# B&R Automation Studio project TD52 (part 139)

#### Vent_ERCyclic.st
```iecst
(*******************************************************************************
Vent_ER			ventilation engine room

This code is confidential and proprietary to the INNIO Company.
It may not be used in any form, or reproduced in any manner,
without the express written permission of the INNIO Company.
Copyright, INNIO Company, 2019

Customized modifications: -
------------------------

History:
-------
V0.1	04.07.1998	Pa			erstellt
 		24.11.1998	Pa			korrekturlesung
V170	06.02.2002	LH			Erfassung Raumtemperatur
V172	02.07.2002	LH			Ventilatoransteuerung, Variante ohne Jalousien
V173	13.11.2002	LH			Einlesen des Analogeinganges in pb17 verlegt
V180	25.02.2003	LH			überarbeitet, Grenzwerte über Rezept
 								Notkühler --> Kühler und erweitert auf 4 Stufen
 								Gemischkühler neu und in 4 Stufen
V181	13.05.2003	LH			Initialisierung für Kühler (Schrittkette)
 		05.06.2003	LH			GW Raumtemperatur angepasst
 		24.06.2003	LH			Gemischkühler in 3 Stufen
V182	04.08.2003	LH			Erfassung Ansauglufttemperatur
V183	25.11.2003	LH			Gemischkühler wieder in 4 Stufen
 								Variante Kombikühler eingeführt
V184	12.01.2004	LH			Ventilation bei Messignal Raumtemperatur
V206	22.06.2004	LH			Raumlüftung NEU aufgrund von Synchronisierproblemen
V207	23.09.2004	LH			20 min. Nachlauf der geregelten Ventilation (Kruckenhauser)
 								Ansauglufttemperatur aktiviert
V2071	05.02.2005	LH			Aktivierung Messtelle Raumtemperatur über Parameter
 		23.02.2005	LH			Nachlauf der geregelten Ventilation nur mit Anforderung Hilfsbetriebe! (Egger)
V2073b	16.05.2006	LH			Lüftung 100% auch bei Gasalarm
V190	09.09.2004	LH			Raumtemperatur und Ansauglufttemperatur --> eigene tasks
 								Lüftung im Stillstand erst mit 40°C
V210	08.09.2004	LH			Variante Raumlüftung für kalte Länder
 								Initialisierung Kühlerschrittkette erweitert auf 11 Regler
 		16.11.2005	LH			Ansteuerung Frequenzumformer bei Gasvoralarm bzw. N2-Spuelung korrigiert
V230	24.01.2008	LH			wegen Einführung Gemischkühlerschrittkette 4-stufigen Gemischkühler gelöscht
V2.34.0	15.10.2008	lettenb.	M_NKWD replaced with M_NKWD_W
V3.10.0	17.02.2010	lettenb.	MRL_FU: EINS -> bAirInVentF(parameter) fehlerbehebung(bruno plattn.)
.								(W2120 störg.raumlüftg.kommt wenn keine raumlüftung)
V3.20.0	30.09.2010	maier(BuR)	M_GSEIN replaced with GCB_ON
.		17.12.2010	lettenb.	purge cycle added, K_var/K_anz/Anz_anfhbt/K_reg setting from parameter
V3.30.0	14.09.2011	lettenb.	FG_FU: dmnd_purge added (bugfix)
V3.99.0 15.02.2013	lettenb.	pb3_VE renamed to Vent_ER
V4.00.0	08.04.2015				FG_FU:(var.with louvers) Para.bER_VentColdCountryMode 'NOT' added(bugfix)
V4.02.0 03.08.2015  Stary       FG_FU: added variant with 2 controlled inlet+outlet louvers
		07.08.2015  Denk		Manual operating auxiliaries control functionality added
		13.08.2015	lettenb.	OUT_VE.tRel_ER_Fan.Do: var.for noFU added(undef.demand ZJAL2 with gcb.on/off)(hackel)
        09.12.2015  Stary       line 189-192: modified variable for louver feedback check
V4.04.0 20.05.2016	lettenb.	tDemPurgeER.Do added, bugfix
V4.04.0 27.09.2016  Stary       Task modified with introduction of cases for the variant-management engine room ventilation
		24.10.2016  Stary       changed parameters for release engine-room ventilation depending on analog position-feedback louvers - bugfix
		21.12.2016  Stary       modification of code after software-test on simulator
		23.01.2017  Stary       modification of code after test with WINMODE (bugfix)
		27.02.2017  Stary       added AND NOT IN_VE.bMsg1031 in release FC (bugfix)
		03.03.2017  lettenb.    added AND NOT IN_VE.bMsg1054 in release FC (bugfix)
		08.05.2017	lettenb.	FG_FU, tRel_ER_FC logic corr., bugfix
V4.05.0 20.09.2017	Messner		Active Cooling Program added
V4.07.0 25.02.2019	lettenb.	bERV_NotRdy engine room ventilation not ready - block engine start added, PWR-FFI-2018-0637 gem. TA 1100-0110
		13.05.2019	lettenb.	ANF_LUE: room vent.active with RTM40(not just minimum fan speed) and extended cooldown time after engine stop
		17.09.2019	lettenb.	ZJAL2: man.aux.control if only 1 inair louver is active, bugfix
V4.10.0	22.12.2020	lettenb.	config VAR.21/22: analog louvers with fix speed fans(set ZJAL1,ZJAL2,AJAL for this config.)
		25.01.2021	lettenb.	engine room ventilation not ready - block engine start: OUT_VE.bERV_NotRdy moved to task MsgVE, bugfix
V4.11.0	23.11.2021	lettenb.	processed signales to AuxRelEngOp (release engine operation) depending on louvers configuration, bugfix
V4.13.0 25.09.2023	Bacci		added IN_VE.tAuxV_Supply_Ok.Di in release FC
		05.12.2023	Bacci		Added ventilation demand before starting the ingition selftest and exhaust scavenging. New DO for inlet louvers demand for customer
V4.14.0 25.11.2024	Bacci		T6 Start procedure with purge start (2024-219): added ventilation demand before purge cranking cycle during fast start preparation
V4.25.0 26.11.2025	Bacci		Safety Function - Insufficient Ventilation (2024-202): reactivation of cold county function and safety plausibility check added

Instructions for use:
--------------------

Outstandings:
------------
*******************************************************************************)
PROGRAM _CYCLIC

	(* parameter *)
	Para.bLouvers;					(* engine room ventilation with louvers *)
	Para.bER_VentColdCountryMode;	(* engine room ventilation cold country mode *)
	Para.bVISA;						(* monitoring according VISA *)

	(*----------------------------------------------------------------------------------------------*)
	(* start ventilation *)
	RTM25 := bT_AirER_Hi1 OR IN_VE.tT_AirER_Ext_Hi1.Di OR IN_VE.bACP_AirER_Dem;

	(* ventilation stage 2 *)
	RTM30 := bT_AirER_Hi2 OR IN_VE.tT_AirER_Ext_Hi2.Di;

	(* start ventilation at stopped engine *)
	RTM40 := bT_AirER_Hi4 OR IN_VE.bACP_AirER_Dem;

	(* demand engine room ventilation for purge cycle *)
	dmnd_purge	:=	Para.bPurgecycle_Active
				AND(IN_VE.bEng_Dem OR IN_VE.bGV_On);

	OUT_VE.tDemPurgeER.Do := dmnd_purge;

	(* signal failure for engine room ventilation *)
	IF Para.bER_VentColdCountryMode THEN
		MS_LUE	:= (IN_VE.bAMM_T_Ch_T1LP_Avg AND IN_VE.bEng_Aux_Dem_CDR)
				OR  MM2VIS.bMsg3152;
	ELSE
		MS_LUE	:=  MM2VIS.bMsg3152;
	END_IF;

	(* purge cycle time *)
	xTON_purgecycle(IN:= OUT_VE.tRel_ER_FC.Do AND NOT MM2VIS.bMsg2120 AND NOT MM2VIS.bMsg2795 AND NOT MM2VIS.bMsg2796, PT:= T#60s);
	OUT_VE.bPurgeER_Rdy := IN_VE.tAirER_FS.Di AND xTON_purgecycle.Q;

	(* Demand engine room ventilation *)
	ANF_LUE	:= IN_VE.bEng_Aux_Dem_CDR
			OR dmnd_purge
			OR IN_VE.bACP_AirER_Dem
			OR RTM40;

	(* fan speed minimum *)
	OUT_VE.tSet_ER_Fan_Min.Do := (IN_VE.bEng_Aux_Dem OR dmnd_purge)
						  AND NOT IN_VE.tGCB_On.Di;

	(* release increased ventilation intensity *)
	IF Para.bInAirER_Fan_FU OR Para.bOutAirER_Fan_FU THEN
		OUT_VE.tRel_ER_Fan.Do := ANF_LUE AND NOT OUT_VE.tSet_ER_Fan_Min.Do;
	ELSE
		OUT_VE.tRel_ER_Fan.Do := ANF_LUE;
	END_IF;

	(* inlet louvers demand for customer. Ventilation in our scope *)
	OUT_VE.tDemERVentInLou_Cust.Do := IN_VE.bInLouDemIgn OR IN_VE.bInLouDemEX OR IN_VE.bInLouDemAG;

	IF IN_VE.bSafetyPLC_Active AND NOT Para.bSafe_ERV_Cust_Active THEN
		(* Cold country mode active for safety PLC *)
		OUT_VE.bERV_ColdCountry := Para.bER_VentColdCountryMode AND NOT (bT_InAirER_LimHi_Lou OR RTM40 OR MS_LUE);

		(*----------------------------------------------------------------*)
		(* safety plausibility check for inlet, outlet louvers and fans *)
		(*----------------------------------------------------------------*)
		(* Minimum release conditions for safety plausibility checks *)
		bRel_ERV_SafeCheck_Min := 	NOT IN_VE.bEng_Aux_Dem_CDR									(* CDR done*)
								AND NOT dmnd_purge												(* Engine room purge done *)
								AND NOT IN_VE.bInLouDemIgn										(* Ignition self test done*)
								AND NOT IN_VE.bInLouDemEX										(* Exhaust gas scavenging done *)
								AND NOT IN_VE.bInLouDemAG										(* Inlet louver demended for purge cycle during fast start preparation *)
								AND NOT (IN_VE.bInAirER_FanSet100 AND IN_VE.bRel_ScavN2)		(* Nitrogen scavenging done*)
								AND NOT IN_VE.bMsg1054											(* No fire alarm *)
								AND NOT IN_VE.bMsg1031											(* No emergency stop*)
								AND NOT IN_VE.bMsg1052											(* No gas prealarm *)
								AND NOT IN_VE.bMsg1053;											(* No gas alarm *)

		(* Extended release conditions for safety plausibility checks *)
		bRel_ERV_SafeCheck_Ext := 		bRel_ERV_SafeCheck_Min
								AND NOT MS_LUE										(* No engine room or engine intake temparture MSF *)
								AND NOT OUT_VE.bMsg2705								(* No engine room differential pressure MSF *)
								AND NOT RTM40										(* High engine room temperature at engine stop *)
								AND NOT IN_VE.tManAuxCtr.bInAirER_Lou1DemOpen 		(* No inlet louvers 1 manual request *)
								AND NOT IN_VE.tManAuxCtr.bInAirER_Lou2DemOpen		(* No inlet louvers 2 manual request *)
								AND NOT IN_VE.tManAuxCtr.bOutAirER_LouDemOpen		(* No outlet louvers manual request *)
								AND NOT IN_VE.tManAuxCtr.bER_FC_Set;				(* No ventilation fan frequency converter manual request *)

		(* engine stopped within 50 min *)
		xTOF_EngStop_SafeCheck(IN:= IN_VE.bEng_Aux_Dem_CDR, PT:= T#50m);

		(* reset plausibility check status *)
		xR_TRIG_bERV_SafeCheck_OK_Rset(CLK := IN_VE.bEng_Aux_Dem_CDR);
		IF xR_TRIG_bERV_SafeCheck_OK_Rset.Q THEN
			bERV_SafeCheck_OK := FALSE;
		END_IF;

		(* General release for safety plauibility checks *)
		bRel_ERV_SafeCheck := (bRel_ERV_SafeCheck_Ext OR (bRel_ERV_SafeCheck_Min AND (NOT xTOF_EngStop_SafeCheck.Q OR IN_VE.bERV_PC_Forced))) AND xOpMode.Stop;
		xR_TRIG_bRel_ERV_SafeCheck(CLK := bRel_ERV_SafeCheck);

		(* break safe plausibility check in case minimum release requirement not fulfilled or extended release not fulfilled while engine stopped within 50 minutes and no check force from safety PLC *)
		IF NOT bRel_ERV_SafeCheck THEN
			iStepCnt_SafeCheck := 0;
		(* activate safe plausibility check in case of extended release conditions fulfilled or minimum release condition fulfilled and engine stopped longer than 50 min or heck force from safety PLC *)
		ELSIF xR_TRIG_bRel_ERV_SafeCheck.Q AND NOT bERV_SafeCheck_OK THEN
			iStepCnt_SafeCheck := 10;
		END_IF;

		(*----------------------------------------------------------------*)
		IF iStepCnt_SafeCheck = 0 THEN
			bERV_SafeCheck_CloseLou	:= FALSE;
			bERV_SafeCheck_OpenLou	:= FALSE;
			OUT_VE.bERV_Lou_PC_OP	:= FALSE;
			OUT_VE.bERV_Lou_PC_CL 	:= FALSE;
			xTON_ERV_SafeCheck_CloseLou(IN:= FALSE, PT:= T#0s);
			xTON_ERV_SafeCheck_OpenLou(IN:= FALSE, PT:= T#0s);
		END_IF;

		(*----------------------------------------------------------------*)
		(* Step 1: close louvers for 3 minutes*)
		IF iStepCnt_SafeCheck = 10 THEN
			bERV_SafeCheck_CloseLou	:= TRUE;
			xTON_ERV_SafeCheck_CloseLou.IN := TRUE;
			xTON_ERV_SafeCheck_CloseLou.PT :=  T#180s;

			IF xTON_ERV_SafeCheck_CloseLou.Q THEN
				bERV_SafeCheck_CloseLou	:= FALSE;
				xTON_ERV_SafeCheck_CloseLou.IN := FALSE;
				xTON_ERV_SafeCheck_CloseLou.PT :=  T#0s;
				iStepCnt_SafeCheck := iStepCnt_SafeCheck + 10;
			END_IF;
		END_IF;
		(*----------------------------------------------------------------*)
		(* Step 2: open louvers for 3 minutes*)
		IF iStepCnt_SafeCheck = 20 THEN
			bERV_SafeCheck_OpenLou	:= TRUE;
			OUT_VE.bERV_Lou_PC_OP := TRUE;
			xTON_ERV_SafeCheck_OpenLou.IN := TRUE;
			xTON_ERV_SafeCheck_OpenLou.PT :=  T#180s;

			IF xTON_ERV_SafeCheck_OpenLou.Q THEN
				bERV_SafeCheck_OpenLou	:= FALSE;
				OUT_VE.bERV_Lou_PC_OP := FALSE;
				xTON_ERV_SafeCheck_OpenLou.IN := TRUE;
				xTON_ERV_SafeCheck_OpenLou.PT :=  T#0s;
				iStepCnt_SafeCheck := iStepCnt_SafeCheck + 10;
			END_IF;
		END_IF;

		(*----------------------------------------------------------------*)
		(* Step 3: close louvers for 3 minutes*)
		IF iStepCnt_SafeCheck = 30 THEN
			bERV_SafeCheck_CloseLou	:= TRUE;
			OUT_VE.bERV_Lou_PC_CL := TRUE;
			xTON_ERV_SafeCheck_CloseLou.IN := TRUE;
			xTON_ERV_SafeCheck_CloseLou.PT :=  T#180s;

			IF xTON_ERV_SafeCheck_CloseLou.Q THEN
				bERV_SafeCheck_CloseLou	:= FALSE;
				OUT_VE.bERV_Lou_PC_CL := FALSE;
				xTON_ERV_SafeCheck_CloseLou.IN := FALSE;
				xTON_ERV_SafeCheck_CloseLou.PT :=  T#0s;
				bERV_SafeCheck_OK := TRUE;
				iStepCnt_SafeCheck := 0;
			END_IF;
		END_IF;

		(*----------------------------------------------------------------*)
	ELSE
		OUT_VE.bERV_ColdCountry :=FALSE;
		bERV_SafeCheck_CloseLou := FALSE;
		bERV_SafeCheck_OpenLou := FALSE;
		OUT_VE.bERV_Lou_PC_OP := FALSE;
		OUT_VE.bERV_Lou_PC_CL := FALSE;
		xTON_ERV_SafeCheck_CloseLou(IN:= FALSE, PT:= T#0s);
		xTON_ERV_SafeCheck_OpenLou(IN:= FALSE, PT:= T#0s);
	END_IF;

		(* Call of the FUB *)
		xTON_ERV_SafeCheck_CloseLou();
		xTON_ERV_SafeCheck_OpenLou();

(*---------------------------------------------------------- INLET LOUVERS HANDLING -----------------------------------------------------------------------------------*)
// 	CONTROL-TYPE
	Para.iTypeCtr_InlLou_ERV; 		// (0-2)  0 ... no control of louvers
							  		//        1 ... engine room inlet louvers 1+2 demanded (DO)
							  		//        2 ... inlet louvers controlled (AO)
//	FEEDBACK-TYPE
	Para.iTypeFeedback_InlLou_ERV; 	// (0-2)  0 ... no feedback-signals
								   	//        1 ... feedback signals digital (DI)
								   	//        2 ... feedback signals analog (AI)

   	(* HANDLING OF CASES FOR RELEASE ROOM-VENTILATION *)
	iValueInlLou := Para.iTypeCtr_InlLou_ERV * 10 + Para.iTypeFeedback_InlLou_ERV; // according to this value the variants will run into the fitting case

	//		0 ... no control and no feedback
	//	   11 ... louvers demanded, feedback signal digital
	//     12 ... louvers demanded, feedback signal analog
	//     21 ... louvers controlled, feedback signal digital
	//     22 ... louvers controlled, feedback signal analog

	CASE iValueInlLou OF

	// ------------------------------------ no control and no feedback -----------------------------------------------------------------------
	  0:
		 	IN_VE.tInAirER_Lou1Opened.Di	:=	IN_VE.tInAirER_Lou1Opened.Di OR	NOT IN_VE.tInAirER_Lou1Opened.GoodQual;
			IN_VE.tInAirER_Lou2Opened.Di	:=	IN_VE.tInAirER_Lou2Opened.Di OR	NOT IN_VE.tInAirER_Lou2Opened.GoodQual;

			(* needed for demand air inlet fan 1 (fix-speed) *)
			ZJAL1 	:=(((bT_InAirER_LimHi_Lou OR NOT Para.bER_VentColdCountryMode) AND (IN_VE.bEng_Aux_Dem_CDR OR dmnd_purge))
					OR	RTM40
					OR	MS_LUE
					OR	IN_VE.bInLouDemIgn (* inlet louver demended for ignition self test *)
					OR	IN_VE.bInLouDemEX  (* inlet louver demended for scavenging *)
					OR	IN_VE.bInLouDemAG  (* inlet louver demended for purge cycle during fast start preparation *)
					OR (IN_VE.bInAirER_FanSet100 AND IN_VE.bRel_ScavN2)
					OR	bERV_SafeCheck_OpenLou) (* louver demand for safety plausibility check*)
					AND NOT bERV_SafeCheck_CloseLou; (* louver closed for safety plausibility check*)

			OUT_VE.tInAirER_Lou1DemOpen.Do	:= (ZJAL1 AND NOT IN_VE.bMsg1054 AND NOT IN_VE.bMsg1031)
											OR	IN_VE.bMsg1052
											OR	IN_VE.bMsg1053;

			(* needed for demand air inlet fan 2 (fix-speed) *)
			IF Para.bInAirER_Fan_FU THEN
				ZJAL2	:=(((bT_InAirER_LimHi_Lou OR NOT Para.bER_VentColdCountryMode) AND (IN_VE.bEng_Aux_Dem_CDR OR dmnd_purge))
						OR	RTM40
						OR	MS_LUE
						OR	IN_VE.bInLouDemIgn (* inlet louver demended for ignition self test *)
						OR	IN_VE.bInLouDemEX  (* inlet louver demended for scavenging *)
						OR	IN_VE.bInLouDemAG  (* inlet louver demended for purge cycle during fast start preparation *)
						OR (IN_VE.bInAirER_FanSet100 AND IN_VE.bRel_ScavN2)
						OR	bERV_SafeCheck_OpenLou) (* louver demand for safety plausibility check*)
						AND NOT bERV_SafeCheck_CloseLou; (* louver closed for safety plausibility check*)

			ELSE
				ZJAL2	:= ((RTM30 AND OUT_VE.tRel_ER_Fan.Do)
						OR	MS_LUE
						OR	IN_VE.bInLouDemIgn (* inlet louver demended for ignition self test *)
						OR	IN_VE.bInLouDemEX  (* inlet louver demended for scavenging *)
						OR	IN_VE.bInLouDemAG  (* inlet louver demended for purge cycle during fast start preparation *)
						OR (IN_VE.bInAirER_FanSet100 AND IN_VE.bRel_ScavN2)
						OR	bERV_SafeCheck_OpenLou) (* louver demand for safety plausibility check*)
						AND NOT bERV_SafeCheck_CloseLou; (* louver closed for safety plausibility check*)
			END_IF;

			OUT_VE.tInAirER_Lou2DemOpen.Do	:= (ZJAL2 AND NOT IN_VE.bMsg1054 AND NOT IN_VE.bMsg1031)
											OR	IN_VE.bMsg1052
											OR	IN_VE.bMsg1053;

			(* release engine room ventilation case 0 *)
			FG_FU_InlLou_Case0	:=	NOT IN_VE.bMsg1054
								AND NOT IN_VE.bMsg1031
								AND	  (((bOMSS_MAT AND IN_VE.bEng_Aux_Dem_CDR)
									OR (bOMSS_MAT AND dmnd_purge)
									OR (bOMSS_MAT AND RTM40)
									OR (bOMSS_MAT AND MM2VIS.bMsg3152)
									OR (IN_VE.bRel_ScavN2 AND IN_VE.bInAirER_FanSet100)
									OR  IN_VE.tManAuxCtr.bER_FC_Set)(* Manual operating auxiliaries control - Handbedienebene *)
									AND NOT bERV_SafeCheck_CloseLou) (* louver /fan off for safety plausibility check*)
									OR IN_VE.bMsg1052
									OR IN_VE.bMsg1053;

	// ------------------------------------- louvers demanded, feedback signal digital -------------------------------------------------------
	 11:
		    (* demand engine room air inlet louver 1 *)
	     	ZJAL1 	:=(((bT_InAirER_LimHi_Lou OR NOT Para.bER_VentColdCountryMode) AND (IN_VE.bEng_Aux_Dem_CDR OR dmnd_purge))
					OR	RTM40
					OR	MS_LUE
					OR (IN_VE.bInAirER_FanSet100 AND IN_VE.bRel_ScavN2)
					OR	IN_VE.bInLouDemIgn (* inlet louver demended for ignition self test *)
					OR	IN_VE.bInLouDemEX  (* inlet louver demended for scavenging *)
					OR	IN_VE.bInLouDemAG  (* inlet louver demended for purge cycle during fast start preparation *)
					OR  IN_VE.tManAuxCtr.bInAirER_Lou1DemOpen			(* Manual operating auxiliaries control - Handbedienebene *)
					OR	bERV_SafeCheck_OpenLou) (* louver demand for safety plausibility check*)
					AND NOT bERV_SafeCheck_CloseLou; (* louver closed for safety plausibility check*)

		 	OUT_VE.tInAirER_Lou1DemOpen.Do	:= (ZJAL1 AND NOT IN_VE.bMsg1054 AND NOT IN_VE.bMsg1031)
											OR	IN_VE.bMsg1052
											OR	IN_VE.bMsg1053;

			(* demand engine room air inlet louver 2 *)
			IF Para.bInAirER_Fan_FU THEN
				ZJAL2	:=(((bT_InAirER_LimHi_Lou OR NOT Para.bER_VentColdCountryMode) AND (IN_VE.bEng_Aux_Dem_CDR OR dmnd_purge))
						OR	RTM40
						OR	MS_LUE
						OR (IN_VE.bInAirER_FanSet100 AND IN_VE.bRel_ScavN2)
						OR	IN_VE.bInLouDemIgn (* inlet louver demended for ignition self test *)
						OR	IN_VE.bInLouDemEX  (* inlet louver demended for scavenging *)
						OR	IN_VE.bInLouDemAG  (* inlet louver demended for purge cycle during fast start preparation *)
						OR (IN_VE.tManAuxCtr.bInAirER_Lou1DemOpen AND NOT Para.bInAirER_Lou2_visible)	(* only 1 inlet louver active *)
						OR  IN_VE.tManAuxCtr.bInAirER_Lou2DemOpen			(* Manual operating auxiliaries control - Handbedienebene *)
						OR	bERV_SafeCheck_OpenLou) (* louver demand for safety plausibility check*)
						AND NOT bERV_SafeCheck_CloseLou; (* louver closed for safety plausibility check*)
			ELSE
				ZJAL2	:= ((RTM30 AND OUT_VE.tRel_ER_Fan.Do)
						OR	MS_LUE
						OR (IN_VE.bInAirER_FanSet100 AND IN_VE.bRel_ScavN2)
						OR	IN_VE.bInLouDemIgn (* inlet louver demended for ignition self test *)
						OR	IN_VE.bInLouDemEX  (* inlet louver demended for scavenging *)
						OR	IN_VE.bInLouDemAG  (* inlet louver demended for purge cycle during fast start preparation *)
						OR (IN_VE.tManAuxCtr.bInAirER_Lou1DemOpen AND NOT Para.bInAirER_Lou2_visible)	(* only 1 inlet louver active *)
						OR  IN_VE.tManAuxCtr.bInAirER_Lou2DemOpen			(* Manual operating auxiliaries control - Handbedienebene *)
						OR	bERV_SafeCheck_OpenLou) (* louver demand for safety plausibility check*)
						AND NOT bERV_SafeCheck_CloseLou; (* louver closed for safety plausibility check*)
			END_IF;

			OUT_VE.tInAirER_Lou2DemOpen.Do	:= (ZJAL2 AND NOT IN_VE.bMsg1054 AND NOT IN_VE.bMsg1031)
											OR	IN_VE.bMsg1052
											OR	IN_VE.bMsg1053;

			(* release engine room ventilation case 11 *)
			IN_VE.tInAirER_Lou2Opened.Di	:=	IN_VE.tInAirER_Lou2Opened.Di OR	NOT IN_VE.tInAirER_Lou2Opened.GoodQual;

			FG_FU_InlLou_Case11 := OUT_VE.tInAirER_Lou1DemOpen.Do AND IN_VE.tInAirER_Lou1Opened.Di
						       AND OUT_VE.tInAirER_Lou2DemOpen.Do AND IN_VE.tInAirER_Lou2Opened.Di;

			FG_InlVent_Step1_CtrInlLou := FALSE; // for correct case-change
			FG_InlVent_Step2_CtrInlLou := FALSE; // for correct case-change

	// ----------------------------------------- louvers demanded, feedback signal analog ----------------------------------------------------
	 12:
			(* demand engine room air inlet louver 1 *)
			ZJAL1 	:=(((bT_InAirER_LimHi_Lou OR NOT Para.bER_VentColdCountryMode) AND (IN_VE.bEng_Aux_Dem_CDR OR dmnd_purge))
					OR	RTM40
					OR	MS_LUE
					OR (IN_VE.bInAirER_FanSet100 AND IN_VE.bRel_ScavN2)
					OR	IN_VE.bInLouDemIgn (* inlet louver demended for ignition self test *)
					OR	IN_VE.bInLouDemEX  (* inlet louver demended for scavenging *)
					OR	IN_VE.bInLouDemAG  (* inlet louver demended for purge cycle during fast start preparation *)
					OR  IN_VE.tManAuxCtr.bInAirER_Lou1DemOpen			(* Manual operating auxiliaries control - Handbedienebene *)
					OR	bERV_SafeCheck_OpenLou) (* louver demand for safety plausibility check*)
					AND NOT bERV_SafeCheck_CloseLou; (* louver closed for safety plausibility check*)

			OUT_VE.tInAirER_Lou1DemOpen.Do	:= (ZJAL1 AND NOT IN_VE.bMsg1054 AND NOT IN_VE.bMsg1031)
											OR	IN_VE.bMsg1052
											OR	IN_VE.bMsg1053;

			(* demand engine room air inlet louver 2 *)
			IF Para.bInAirER_Fan_FU THEN
				ZJAL2	:=(((bT_InAirER_LimHi_Lou OR NOT Para.bER_VentColdCountryMode) AND (IN_VE.bEng_Aux_Dem_CDR OR dmnd_purge))
						OR	RTM40
						OR	MS_LUE
						OR (IN_VE.bInAirER_FanSet100 AND IN_VE.bRel_ScavN2)
						OR	IN_VE.bInLouDemIgn (* inlet louver demended for ignition self test *)
						OR	IN_VE.bInLouDemEX  (* inlet louver demended for scavenging *)
						OR	IN_VE.bInLouDemAG  (* inlet louver demended for purge cycle during fast start preparation *)
						OR (IN_VE.tManAuxCtr.bInAirER_Lou1DemOpen AND NOT Para.bInAirER_Lou2_visible)	(* only 1 inlet louver active *)
						OR  IN_VE.tManAuxCtr.bInAirER_Lou2DemOpen			(* Manual operating auxiliaries control - Handbedienebene *)
						OR	bERV_SafeCheck_OpenLou) (* louver demand for safety plausibility check*)
						AND NOT bERV_SafeCheck_CloseLou; (* louver closed for safety plausibility check*)
			ELSE
				ZJAL2	:= ((RTM30 AND OUT_VE.tRel_ER_Fan.Do)
						OR	MS_LUE
						OR (IN_VE.bInAirER_FanSet100 AND IN_VE.bRel_ScavN2)
						OR	IN_VE.bInLouDemIgn (* inlet louver demended for ignition self test *)
						OR	IN_VE.bInLouDemEX  (* inlet louver demended for scavenging *)
						OR	IN_VE.bInLouDemAG  (* inlet louver demended for purge cycle during fast start preparation *)
						OR (IN_VE.tManAuxCtr.bInAirER_Lou1DemOpen AND NOT Para.bInAirER_Lou2_visible)	(* only 1 inlet louver active *)
						OR  IN_VE.tManAuxCtr.bInAirER_Lou2DemOpen			(* Manual operating auxiliaries control - Handbedienebene *)
						OR	bERV_SafeCheck_OpenLou) (* louver demand for safety plausibility check*)
						AND NOT bERV_SafeCheck_CloseLou; (* louver closed for safety plausibility check*)
			END_IF;

			OUT_VE.tInAirER_Lou2DemOpen.Do	:= (ZJAL2 AND NOT IN_VE.bMsg1054 AND NOT IN_VE.bMsg1031)
											OR	IN_VE.bMsg1052
											OR	IN_VE.bMsg1053;

			(* check of position from inlet-louvers *)
			xGR_MAXR_InlLou1(In := IN_VE.tPos_InlLou1.Ai, Gw := Para.rPosLim_InlLou_Rel_ERV, Hy := Para.rPosLim_InlLou_Rel_ERV_Hy);
			xGR_MAXR_InlLou2(In := IN_VE.tPos_InlLou2.Ai, Gw := Para.rPosLim_InlLou_Rel_ERV, Hy := Para.rPosLim_InlLou_Rel_ERV_Hy);

			Pos_InlLou1_OK := Para.bPos_InlLou1_Active AND xGR_MAXR_InlLou1.Q;
			Pos_InlLou2_OK := Para.bPos_InlLou2_Active AND xGR_MAXR_InlLou2.Q;
			OUT_VE.Pos_InlLou1_OK := Pos_InlLou1_OK; // for release auxiliaries --> monitoring A1129 (AG)
			OUT_VE.Pos_InlLou2_OK := Pos_InlLou2_OK; // for release auxiliaries --> monitoring A1129 (AG)

			(* release engine room ventilation case 12 *)
			FG_FU_InlLou_Case12   := (OUT_VE.tInAirER_Lou1DemOpen.Do AND Pos_InlLou1_OK)
								AND ((OUT_VE.tInAirER_Lou2DemOpen.Do AND Pos_InlLou2_OK) OR NOT Para.bPos_InlLou2_Active);

			FG_InlVent_Step1_CtrInlLou := FALSE; // for correct case-change
			FG_InlVent_Step2_CtrInlLou := FALSE; // for correct case-change

	// -------------------------------------- louvers controlled, feedback signal digital --------------------------------------------------------------------
	 21:
			(* demand engine room air inlet louver *)
			ZJAL1 	:=((IN_VE.bEng_Aux_Dem_CDR OR dmnd_purge)
					OR	RTM40
					OR	MS_LUE
					OR (IN_VE.bInAirER_FanSet100 AND IN_VE.bRel_ScavN2)
					OR	bERV_SafeCheck_OpenLou) (* louver demand for safety plausibility check*)
					AND NOT bERV_SafeCheck_CloseLou; (* louver closed for safety plausibility check*)
					(*OUT_IG.bInLouDemIgn AND OUT_IG.bInLouDemEX AND IN_VE.bInLouDemAG not needed for fan activation. Louver AO signal defined in the Ctr_InlLou*)

			ZJAL2	:= ((RTM30 AND OUT_VE.tRel_ER_Fan.Do)
					OR	MS_LUE
					OR (IN_VE.bInAirER_FanSet100 AND IN_VE.bRel_ScavN2)
					OR	bERV_SafeCheck_OpenLou) (* louver demand for safety plausibility check*)
					AND NOT bERV_SafeCheck_CloseLou; (* louver closed for safety plausibility check*)

			(* release engine room ventilation case 21 *)
			IN_VE.tInAirER_Lou2Opened.Di := IN_VE.tInAirER_Lou2Opened.Di OR	NOT IN_VE.tInAirER_Lou2Opened.GoodQual;

			FG_FU_InlLou_Case21   := Para.bCtr_InlLou AND IN_VE.tInAirER_Lou1Opened.Di AND IN_VE.tInAirER_Lou2Opened.Di;

			(* air inlet fan 1 *)
			Release_InlVent_Step1_INT := (ZJAL1 AND NOT IN_VE.bMsg1054 AND NOT IN_VE.bMsg1031)  // general release ventilation step 1 depending on temperature, gas-alarm etc.
									OR	IN_VE.bMsg1052
									OR	IN_VE.bMsg1053;
			FG_InlVent_Step1_CtrInlLou := Release_InlVent_Step1_INT AND Para.bCtr_InlLou AND IN_VE.tInAirER_Lou1Opened.Di; 	// fix-speed inlet-fan 1

			(* air inlet fan 2 *)
			Release_InlVent_Step2_INT := (ZJAL2 AND NOT IN_VE.bMsg1054 AND NOT IN_VE.bMsg1031)  // general release ventilation step 2 depending on temperature, gas-alarm etc.
									OR	IN_VE.bMsg1052
									OR	IN_VE.bMsg1053;
			FG_InlVent_Step2_CtrInlLou := Release_InlVent_Step2_INT AND Para.bCtr_InlLou AND IN_VE.tInAirER_Lou1Opened.Di AND IN_VE.tInAirER_Lou2Opened.Di;  // fix-speed inlet-fan 2

			OUT_VE.tInAirER_Lou1DemOpen.Do := FALSE; // for correct case-change
			OUT_VE.tInAirER_Lou2DemOpen.Do := FALSE; // for correct case-change

	// --------------------------------------- louvers controlled, feedback signal analog ---------------------------------------------------------------------
	 22:
			(* demand engine room air inlet louver *)
			ZJAL1 	:=((IN_VE.bEng_Aux_Dem_CDR OR dmnd_purge)
					OR	RTM40
					OR	MS_LUE
					OR (IN_VE.bInAirER_FanSet100 AND IN_VE.bRel_ScavN2)
					OR	bERV_SafeCheck_OpenLou) (* louver demand for safety plausibility check*)
					AND NOT bERV_SafeCheck_CloseLou; (* louver closed for safety plausibility check*)
					(*OUT_IG.bInLouDemIgn AND OUT_IG.bInLouDemEX AND IN_VE.bInLouDemAG not needed for fan activation. Louver AO signalo defined in the Ctr_InlLou*)

			ZJAL2	:= ((RTM30 AND OUT_VE.tRel_ER_Fan.Do)
					OR	MS_LUE
					OR (IN_VE.bInAirER_FanSet100 AND IN_VE.bRel_ScavN2)
					OR	bERV_SafeCheck_OpenLou) (* louver demand for safety plausibility check*)
					AND NOT bERV_SafeCheck_CloseLou; (* louver closed for safety plausibility check*)

			(* check of position from inlet-louvers *)
			xGR_MAXR_InlLou1(In := IN_VE.tPos_InlLou1.Ai, Gw := Para.rPosLim_InlLou_Rel_ERV, Hy := Para.rPosLim_InlLou_Rel_ERV_Hy);
			xGR_MAXR_InlLou2(In := IN_VE.tPos_InlLou2.Ai, Gw := Para.rPosLim_InlLou_Rel_ERV, Hy := Para.rPosLim_InlLou_Rel_ERV_Hy);

			Pos_InlLou1_OK := Para.bPos_InlLou1_Active AND xGR_MAXR_InlLou1.Q;
			Pos_InlLou2_OK := Para.bPos_InlLou2_Active AND xGR_MAXR_InlLou2.Q;
			OUT_VE.Pos_InlLou1_OK := Pos_InlLou1_OK; // for release auxiliaries --> monitoring A1129 (AG)
			OUT_VE.Pos_InlLou2_OK := Pos_InlLou2_OK; // for release auxiliaries --> monitoring A1129 (AG)

			(* release engine room ventilation CASE 22 *)
			FG_FU_InlLou_Case22   := Para.bCtr_InlLou AND Pos_InlLou1_OK AND (Pos_InlLou2_OK OR NOT Para.bPos_InlLou2_Active);

			(* air inlet fan 1 *)
			Release_InlVent_Step1_INT := (ZJAL1 AND NOT IN_VE.bMsg1054 AND NOT IN_VE.bMsg1031)  // general release ventilation step 1 depending on temperature, gas-alarm etc.
									OR	IN_VE.bMsg1052
									OR	IN_VE.bMsg1053;
			FG_InlVent_Step1_CtrInlLou := Release_InlVent_Step1_INT AND Para.bCtr_InlLou AND Pos_InlLou1_OK;  // fix-speed inlet-fan 1

			(* air inlet fan 2 *)
			Release_InlVent_Step2_INT := (ZJAL2 AND NOT IN_VE.bMsg1054 AND NOT IN_VE.bMsg1031)  // general release ventilation step 2 depending on temperature, gas-alarm etc.
									OR	IN_VE.bMsg1052
									OR	IN_VE.bMsg1053;
			FG_InlVent_Step2_CtrInlLou := Release_InlVent_Step2_INT AND Para.bCtr_InlLou AND Pos_InlLou1_OK AND (Pos_InlLou2_OK OR NOT Para.bPos_InlLou2_Active);  // fix-speed inlet-fan 2

			OUT_VE.tInAirER_Lou1DemOpen.Do := FALSE; // for correct case-change
			OUT_VE.tInAirER_Lou2DemOpen.Do := FALSE; // for correct case-change

	END_CASE;

(*---------------------------------------------------------- OUTLET LOUVERS HANDLING -----------------------------------------------------------------------------------*)
// 	CONTROL-TYPE
	Para.iTypeCtr_OutlLou_ERV; 		// (0-2)  0 ... no control of louvers
							   		//        1 ... engine room outlet louvers 1+2 demanded (DO)
							   		//        2 ... outlet louvers controlled (AO)
//	FEEDBACK-TYPE
	Para.iTypeFeedback_OutlLou_ERV; // (0-2)  0 ... no feedback-signals
									//        1 ... feedback signals digital (DI)
									//        2 ... feedback signals analog (AI)

	(* HANDLING OF CASES FOR RELEASE ROOM-VENTILATION *)
	iValueOutlLou := Para.iTypeCtr_OutlLou_ERV*10 + Para.iTypeFeedback_OutlLou_ERV; // according to this value the variants will run into the fitting case

	//		0 ... no control and no feedback
	//	   11 ... louvers demanded, feedback signal digital
	//     12 ... louvers demanded, feedback signal analog
	//     21 ... louvers controlled, feedback signal digital
	//     22 ... louvers controlled, feedback signal analog

	CASE iValueOutlLou OF

		// --------------------------------------- no control and no feedback ------------------------------------------------------------
		0:
				IN_VE.tOutAirER_LouOpened.Di := IN_VE.tOutAirER_LouOpened.Di OR	NOT IN_VE.tOutAirER_LouOpened.GoodQual;

				(* needed for demand air inlet fan 1+2 (fix-speed) *)
				AJAL	:=	(IN_VE.bEng_Aux_Dem_CDR
						OR	dmnd_purge
						OR	RTM40
						OR	MS_LUE
						OR (IN_VE.bInAirER_FanSet100 AND IN_VE.bRel_ScavN2)
						OR	bERV_SafeCheck_OpenLou) (* louver demand for safety plausibility check*)
						AND NOT bERV_SafeCheck_CloseLou; (* louver closed for safety plausibility check*)

				OUT_VE.tOutAirER_LouDemOpen.Do	:= (AJAL AND NOT IN_VE.bMsg1031 AND NOT IN_VE.bMsg1054)
												OR	IN_VE.bMsg1052
												OR	IN_VE.bMsg1053;

				(* release engine room ventilation case 0 *)
				FG_FU_OutLou_Case0	:=	NOT IN_VE.bMsg1054
									AND NOT IN_VE.bMsg1031
									AND	  (((bOMSS_MAT AND IN_VE.bEng_Aux_Dem_CDR)
										OR (bOMSS_MAT AND dmnd_purge)
										OR (bOMSS_MAT AND RTM40)
										OR (bOMSS_MAT AND MM2VIS.bMsg3152)
										OR (IN_VE.bRel_ScavN2 AND IN_VE.bInAirER_FanSet100)
										OR  IN_VE.tManAuxCtr.bER_FC_Set) (* Manual operating auxiliaries control - Handbedienebene *)
										AND NOT bERV_SafeCheck_CloseLou) (* louver /fan off for safety plausibility check*)
										OR IN_VE.bMsg1052
										OR IN_VE.bMsg1053;

	// ---------------------------------------louvers demanded, feedback signal digital -----------------------------------------------------------
		11:
				(* demand engine room air outlet louvers *)
				AJAL	:=	(IN_VE.bEng_Aux_Dem_CDR
						OR	dmnd_purge
						OR	RTM40
						OR	MS_LUE
						OR (IN_VE.bInAirER_FanSet100 AND IN_VE.bRel_ScavN2)
						OR  IN_VE.tManAuxCtr.bOutAirER_LouDemOpen			(* Manual operating auxiliaries control - Handbedienebene *)
						OR	bERV_SafeCheck_OpenLou) (* louver demand for safety plausibility check*)
						AND NOT bERV_SafeCheck_CloseLou; (* louver closed for safety plausibility check*)

				OUT_VE.tOutAirER_LouDemOpen.Do	:= (AJAL AND NOT IN_VE.bMsg1031 AND NOT IN_VE.bMsg1054)
												OR	IN_VE.bMsg1052
												OR	IN_VE.bMsg1053;

				(* Release engine room ventilation case 12 *)
				FG_FU_OutlLou_Case11 := OUT_VE.tOutAirER_LouDemOpen.Do AND IN_VE.tOutAirER_LouOpened.Di;

				FG_InlVent_Step12_CtrOutlLou := FALSE; // for correct case-change

	// ---------------------------------------- louvers demanded, feedback signal analog -----------------------------------------------------------
		12:
				(* demand engine room air outlet louvers *)
				AJAL	:=	(IN_VE.bEng_Aux_Dem_CDR
						OR	dmnd_purge
						OR	RTM40
						OR	MS_LUE
						OR (IN_VE.bInAirER_FanSet100 AND IN_VE.bRel_ScavN2)
						OR  IN_VE.tManAuxCtr.bOutAirER_LouDemOpen			(* Manual operating auxiliaries control - Handbedienebene *)
						OR	bERV_SafeCheck_OpenLou) (* louver demand for safety plausibility check*)
						AND NOT bERV_SafeCheck_CloseLou; (* louver closed for safety plausibility check*)

				OUT_VE.tOutAirER_LouDemOpen.Do	:= (AJAL AND NOT IN_VE.bMsg1031 AND NOT IN_VE.bMsg1054)
												OR	IN_VE.bMsg1052
												OR	IN_VE.bMsg1053;

				(* check of position from outlet-louvers *)
				xGR_MAXR_OutlLou1(In:= IN_VE.tPos_OutlLou1.Ai, Gw:= Para.rPosLim_OutlLou_Rel_ERV, Hy:= Para.rPosLim_OutlLou_Rel_ERV_Hy);
				xGR_MAXR_OutlLou2(In:= IN_VE.tPos_OutlLou2.Ai, Gw:= Para.rPosLim_OutlLou_Rel_ERV, Hy:= Para.rPosLim_OutlLou_Rel_ERV_Hy);

				Pos_OutlLou1_OK := Para.bPos_OutlLou1_Active AND xGR_MAXR_OutlLou1.Q;
				Pos_OutlLou2_OK := Para.bPos_OutlLou2_Active AND xGR_MAXR_OutlLou2.Q;
				OUT_VE.Pos_OutlLou1_OK := Pos_OutlLou1_OK; // for release auxiliaries --> monitoring A1129 (AG)
				OUT_VE.Pos_OutlLou2_OK := Pos_OutlLou2_OK; // for release auxiliaries --> monitoring A1129 (AG)

				(* release engine room ventilation case 12 *)
				FG_FU_OutlLou_Case12	:= OUT_VE.tOutAirER_LouDemOpen.Do AND Pos_OutlLou1_OK AND (Pos_OutlLou2_OK OR NOT Para.bPos_OutlLou2_Active);

				FG_InlVent_Step12_CtrOutlLou := FALSE; // for correct case-change

	// ------------------------------------------- louvers controlled, feedback signal digital ---------------------------------------------------------
		21:
				(* demand air inlet fan 1+2 (fix-speed) *)
				AJAL	:=	(IN_VE.bEng_Aux_Dem_CDR
						OR	dmnd_purge
						OR	RTM40
						OR	MS_LUE
						OR (IN_VE.bInAirER_FanSet100 AND IN_VE.bRel_ScavN2)
						OR	bERV_SafeCheck_OpenLou) (* louver demand for safety plausibility check*)
						AND NOT bERV_SafeCheck_CloseLou; (* louver closed for safety plausibility check*)

				(* release engine room ventilation case 21 *)
				FG_FU_OutlLou_Case21	:= (Para.bCtr_OutlLou_RDP OR Para.bCtr_OutlLou_RT) AND IN_VE.tOutAirER_LouOpened.Di;

				(* air inlet fan 1+2 *)
			    Release_InlVent_StepINT	:= (AJAL AND NOT IN_VE.bMsg1031 AND NOT IN_VE.bMsg1054)	// general release ventilation step 1 depending on temperature, gas-alarm etc.
										OR	IN_VE.bMsg1052
										OR	IN_VE.bMsg1053;
				FG_InlVent_Step12_CtrOutlLou := Release_InlVent_StepINT AND (Para.bCtr_OutlLou_RDP OR Para.bCtr_OutlLou_RT) AND IN_VE.tOutAirER_LouOpened.Di;  // fix-speed inlet-fan 1+2

				OUT_VE.tOutAirER_LouDemOpen.Do := FALSE; // for correct case-change

	// -------------------------------------------- louvers controlled, feedback signal analog ---------------------------------------------------------
		22:
				(* demand air inlet fan 1+2 (fix-speed) *)
				AJAL	:=	(IN_VE.bEng_Aux_Dem_CDR
						OR	dmnd_purge
						OR	RTM40
						OR	MS_LUE
						OR (IN_VE.bInAirER_FanSet100 AND IN_VE.bRel_ScavN2)
						OR	bERV_SafeCheck_OpenLou) (* louver demand for safety plausibility check*)
						AND NOT bERV_SafeCheck_CloseLou; (* louver closed for safety plausibility check*)

				(* check of position from outlet-louvers *)
				xGR_MAXR_OutlLou1(In:= IN_VE.tPos_OutlLou1.Ai, Gw:= Para.rPosLim_OutlLou_Rel_ERV, Hy:= Para.rPosLim_OutlLou_Rel_ERV_Hy);
				xGR_MAXR_OutlLou2(In:= IN_VE.tPos_OutlLou2.Ai, Gw:= Para.rPosLim_OutlLou_Rel_ERV, Hy:= Para.rPosLim_OutlLou_Rel_ERV_Hy);

				Pos_OutlLou1_OK := Para.bPos_OutlLou1_Active AND xGR_MAXR_OutlLou1.Q;
				Pos_OutlLou2_OK := Para.bPos_OutlLou2_Active AND xGR_MAXR_OutlLou2.Q;
				OUT_VE.Pos_OutlLou1_OK := Pos_OutlLou1_OK; // for release auxiliaries --> monitoring A1129 (AG)
				OUT_VE.Pos_OutlLou2_OK := Pos_OutlLou2_OK; // for release auxiliaries --> monitoring A1129 (AG)

				(* release engine room ventilation CASE 22 *)
				FG_FU_OutlLou_Case22	:= (Para.bCtr_OutlLou_RDP OR Para.bCtr_OutlLou_RT) AND Pos_OutlLou1_OK AND (Pos_OutlLou2_OK OR NOT Para.bPos_OutlLou2_Active);

				(* air inlet fan 1+2 *)
				Release_InlVent_StepINT	:= (AJAL AND NOT IN_VE.bMsg1031 AND NOT IN_VE.bMsg1054)	// general release ventilation step 1 depending on temperature, gas-alarm etc.
										OR	IN_VE.bMsg1052
										OR	IN_VE.bMsg1053;
				FG_InlVent_Step12_CtrOutlLou := Release_InlVent_StepINT AND (Para.bCtr_OutlLou_RDP OR Para.bCtr_OutlLou_RT)
											AND Pos_OutlLou1_OK AND (Pos_OutlLou2_OK OR NOT Para.bPos_OutlLou2_Active);	// fix-speed inlet-fan 1+2

				OUT_VE.tOutAirER_LouDemOpen.Do := FALSE; // for correct case-change

	END_CASE;

(*------------------------ CASE CHECK FOR RELEASE ENGINE ROOM VENTILATION -----------------------------------------*)
	(* Inlet ventilation *)
	FG_FU_InlLou_ZW := (FG_FU_InlLou_Case0  AND iValueInlLou = 0)
					OR (FG_FU_InlLou_Case11 AND iValueInlLou = 11)
					OR (FG_FU_InlLou_Case12 AND iValueInlLou = 12)
					OR (FG_FU_InlLou_Case21 AND iValueInlLou = 21)
					OR (FG_FU_InlLou_Case22 AND iValueInlLou = 22);

	(* Outlet ventilation *)
	FG_FU_OutlLou_ZW := (FG_FU_OutLou_Case0  AND iValueOutlLou = 0)
					 OR (FG_FU_OutlLou_Case11 AND iValueOutlLou = 11)
					 OR (FG_FU_OutlLou_Case12 AND iValueOutlLou = 12)
					 OR (FG_FU_OutlLou_Case21 AND iValueOutlLou = 21)
					 OR (FG_FU_OutlLou_Case22 AND iValueOutlLou = 22);

(*---------------------------------------------------------- ROOM VENTILATION FAN HANDLING -----------------------------------------------------------------------------------*)

		(* air inlet fan 1 *)
		OUT_VE.tInAirER_Fan1DemOn.Do :=	(((OUT_VE.tInAirER_Lou1DemOpen.Do OR IN_VE.tManAuxCtr.bInAirER_Fan1DemOn) AND IN_VE.tInAirER_Lou1Opened.Di) OR FG_InlVent_Step1_CtrInlLou)
									AND (((OUT_VE.tOutAirER_LouDemOpen.Do OR IN_VE.tManAuxCtr.bInAirER_Fan1DemOn) AND IN_VE.tOutAirER_LouOpened.Di) OR FG_InlVent_Step12_CtrOutlLou);

		(* air inlet fan 2 *)
		OUT_VE.tInAirER_Fan2DemOn.Do := (((OUT_VE.tInAirER_Lou2DemOpen.Do OR IN_VE.tManAuxCtr.bInAirER_Fan2DemOn) AND IN_VE.tInAirER_Lou2Opened.Di) OR FG_InlVent_Step2_CtrInlLou)
									AND (((OUT_VE.tOutAirER_LouDemOpen.Do OR IN_VE.tManAuxCtr.bInAirER_Fan2DemOn) AND IN_VE.tOutAirER_LouOpened.Di) OR FG_InlVent_Step12_CtrOutlLou);

		(* release frequency converter for engine room ventilation (inlet/outlet) *)

		IF IN_VE.tManAuxCtr.bER_FC_Set THEN				(* Manual operating auxiliaries control - Handbedienebene *)
			FG_FU	:=	NOT IN_VE.bMsg1031
					AND NOT IN_VE.bMsg1054
					AND		FG_FU_InlLou_ZW
					AND 	FG_FU_OutlLou_ZW
					AND		IN_VE.tAuxV_Supply_Ok.Di;
		ELSE
			FG_FU	:=	NOT IN_VE.bMsg1031
					AND NOT IN_VE.bMsg1054
					AND		FG_FU_InlLou_ZW
					AND 	FG_FU_OutlLou_ZW
					AND		IN_VE.tAuxV_Supply_Ok.Di;
		END_IF;
		OUT_VE.tRel_ER_FC.Do := FG_FU OR IN_VE.bMsg1052 OR IN_VE.bMsg1053 OR (IN_VE.bACP_AirER_Dem AND NOT bERV_SafeCheck_CloseLou);

		(* demand fixed fan speed *)
		FU_FIX		:=     (MS_LUE AND OUT_VE.tRel_ER_Fan.Do)
					OR		bT_AirER_Hi
					OR	NOT	IN_VE.tT_AirER_Ext_Hi.Di
					OR 	   (IN_VE.bInAirER_FanSet100 AND IN_VE.bRel_ScavN2)
					OR		IN_VE.bMsg1052 OR IN_VE.bMsg1053;

		bCtrER_YFix := OUT_VE.tRel_ER_FC.Do AND FU_FIX;

(*---------------------------------------------------------------------------*)
	(* release engine room temperature controller *)
	(* see task: Ctr_ER *)
(*---------------------------------------------------------------------------*)
	(* open or not closed inlet louvers release from ventilation for ignition and exhaust*)
	IF iValueInlLou =0 THEN
		OUT_VE.bInLouRelVE := IN_VE.tInAirER_Lou1Opened.Di OR IN_VE.tInAirER_Lou2Opened.Di;
	ELSE
		OUT_VE.bInLouRelVE := (IN_VE.tInAirER_Lou1Opened.Di AND IN_VE.tInAirER_Lou1Opened.GoodQual) OR ((NOT IN_VE.tInAirER_Lou1Closed.Di) AND IN_VE.tInAirER_Lou1Closed.GoodQual) OR
							  (Pos_InlLou1_OK AND IN_VE.tPos_InlLou1.GoodQual) OR
							  (IN_VE.tInAirER_Lou2Opened.Di AND IN_VE.tInAirER_Lou2Opened.GoodQual) OR ((NOT IN_VE.tInAirER_Lou2Closed.Di) AND IN_VE.tInAirER_Lou2Closed.GoodQual) OR
							  (Pos_InlLou2_OK AND IN_VE.tPos_InlLou2.GoodQual);
	END_IF;

(*---------------------------------------------------------------------------*)
	(* processed signales to AuxRelEngOp (release engine operation) depending on louvers configuration *)
	OUT_VE.tInAirER_Lou1Opened.Di := IN_VE.tInAirER_Lou1Opened.Di;
	OUT_VE.tInAirER_Lou2Opened.Di := IN_VE.tInAirER_Lou2Opened.Di;
	OUT_VE.tOutAirER_LouOpened.Di := IN_VE.tOutAirER_LouOpened.Di;

END_PROGRAM
```

#### Vent_ER.var
```iecst
VAR
	xTON_purgecycle : TON := (0);
	xGR_MAXR_InlLou2 : GR_MAXR := (0); (*minimum opening position of inlet louver 2 for release FQ room ventilation*)
	xGR_MAXR_InlLou1 : GR_MAXR := (0); (*minimum opening position of inlet louver 1 for release FQ room ventilation*)
	xGR_MAXR_OutlLou1 : GR_MAXR := (0); (*minimum opening position of outlet louver 1 for release FQ room ventilation*)
	xGR_MAXR_OutlLou2 : GR_MAXR := (0); (*minimum opening position of outlet louver 2 for release FQ room ventilation*)
	FG_FU_InlLou_Case22 : BOOL; (*Release FQ roomventilation with controlled inlet louvers and analog feedback signal*)
	FG_FU_InlLou_Case21 : BOOL; (*Release FQ roomventilation with controlled inlet louvers and digital feedback signal*)
	FG_FU_InlLou_Case12 : BOOL; (*Release FQ roomventilation with demanded inlet louvers and analog feedback-signal*)
	FG_FU_InlLou_Case11 : BOOL; (*Release FQ roomventilation with demanded inlet louvers and digital feedback-signal*)
	FG_FU_InlLou_Case0 : BOOL; (*Release FQ roomventilation - no inlet louvers control existing*)
	FG_FU_OutlLou_Case22 : BOOL; (*Release FQ roomventilation with controlled outlet louvers and analog feedback signal*)
	FG_FU_OutlLou_Case21 : BOOL; (*Release FQ roomventilation with controlled outlet louvers and digital feedback signal*)
	FG_FU_OutlLou_Case12 : BOOL; (*Release FQ roomventilation with demanded outlet louver and analog feedback-signal*)
	FG_FU_OutlLou_Case11 : BOOL; (*Release FQ roomventilation with demanded outlet louver and digital feedback-signal*)
	FG_FU_OutLou_Case0 : BOOL; (*Release FQ roomventilation - no outlet louvers control existing*)
	FG_FU_OutlLou_ZW : BOOL; (*intern value release outlet ventilation*)
	FG_FU_InlLou_ZW : BOOL; (*intern value release inlet ventilation*)
	FG_InlVent_Step12_CtrOutlLou : BOOL := 0; (*release for fix-speed inlet-fan 1+2 depending on ctr outlet louver*)
	FG_InlVent_Step2_CtrInlLou : BOOL := 0; (*release for fix-speed inlet-fan 2 depending on ctr inlet louver*)
	FG_InlVent_Step1_CtrInlLou : BOOL := 0; (*release for fix-speed inlet-fan 1 depending on ctr inlet louver*)
	Release_InlVent_StepINT : BOOL := 0; (*general release ventilation step 1+2 depending on temperature, gas-alarm etc.*)
	Release_InlVent_Step2_INT : BOOL := 0; (*general release ventilation step 2 depending on temperature, gas-alarm etc.*)
	Release_InlVent_Step1_INT : BOOL := 0; (*general release ventilation step 1 depending on temperature, gas-alarm etc.*)
	bRel_ERV_SafeCheck_Min : BOOL; (*Minimum release conditions for safety plausibility checks *)
	bRel_ERV_SafeCheck_Ext : BOOL; (*Extended release conditions for safety plausibility checks *)
	xTOF_EngStop_SafeCheck : TOF; (*Engine stop timer for safety plausibility checks*)
	bERV_SafeCheck_OK : BOOL; (*Safety plausibility checks executed*)
	iStepCnt_SafeCheck : INT; (*Safety plausibility checks step counter*)
	xTON_ERV_SafeCheck_CloseLou : TON; (*Safety plausibility checks close louver timer*)
	xTON_ERV_SafeCheck_OpenLou : TON; (*Safety plausibility checks open louver timer*)
	bRel_ERV_SafeCheck : BOOL; (*Safety plausibility checks released*)
	xR_TRIG_bRel_ERV_SafeCheck : R_TRIG; (*Safety plausibility checks released positive edge*)
	xR_TRIG_bERV_SafeCheck_OK_Rset : R_TRIG; (*Safety plausibility checks executed reset*)
END_VAR
```

### Program Logical/Ventilation/T_InAirER (IEC, version 4.04.0) - engine room air inlet temperature 

#### T_InAirERCyclic.st
```iecst
(*******************************************************************************
T_InAirER		temperature inlet air engine room

This code is confidential and proprietary to the INNIO Company.
It may not be used in any form, or reproduced in any manner,
without the express written permission of the INNIO Company.
Copyright, INNIO Company, 2019

Customized modifications: -
------------------------

History:
-------
V190	12.08.2004	LH			erstellt
V220	01.03.2007	LH			Erweiterung auf Pt100
 		10.04.2007	LH			Korrektur Messignalüberwachung, Zuweisung für Pt100
V2201	23.07.2007	LH			Messignalüberwachung: UGR -20°C --> -50°C
V3.99.0	22.02.2013	lettenb.	a_lt renamed to T_InAirER, p_limitVE included
		26.04.2013				xGRMAX_T_InAirER_LimHi: Hy 10.0 --> 1.0 bugfix
		02.10.2013				rP_Red_T_InAirER_Lim  := 0.0; bugfix
V4.04	02.11.2016	Tinello		monitoring "bT_InAirER_Hi" deleted, Para.bT_InAirER_Active removed --> moved to modul CH

Instructions for use:
--------------------
Outstandings:
------------
*******************************************************************************)
PROGRAM _CYCLIC

	(*---------------------------------------------------------------------------*)
	(* engine room inlet air temperature high (open inlet louvers) *)
	IN_VE.rT_Ch_T1LP_Avg;	(* value(from CH) = 0 in case of no sensor is active or signal failure *)

	xGRMAX_T_InAirER_LimHi_Lou(Gw:= Para.rT_InAirER_LimHi_Lou, Hy:= Para.rT_Lou_InAirER_HyHi, In:= IN_VE.rT_Ch_T1LP_Avg);
	bT_InAirER_LimHi_Lou := IN_VE.tPB2MM.bParaSetupOk AND xGRMAX_T_InAirER_LimHi_Lou.Q;

	(*---------------------------------------------------------------------------*)
	(* engine room inlet air temperature high (start fan *)
	xGRMAX_T_InAirER_LimHi_Fan(Gw:= Para.rT_InAirER_LimHi_Fan, Hy:= Para.rT_Fan_InAirER_HyHi, In:= IN_VE.rT_Ch_T1LP_Avg);
	bT_InAirER_LimHi_Fan := IN_VE.tPB2MM.bParaSetupOk AND xGRMAX_T_InAirER_LimHi_Fan.Q;

	(*===========================================================================*)
	(* power limitation by engine room air inlet temperature high from engine nominal power *)
	IF Para.bPred_T_InAirER_Active THEN
		IF Para.rT_Pred_InAirER_Start2 > Para.rT_Pred_InAirER_Start THEN	(* parameter plausibility check *)
			rT_Pred_InAirER_Start1	:=	Para.rT_Pred_InAirER_Start;			(* copy to local pv *)
			rT_Pred_InAirER_Rate1	:=	Para.rT_Pred_InAirER_Rate;
			rT_Pred_InAirER_Start2	:=	Para.rT_Pred_InAirER_Start2;
			rT_Pred_InAirER_Rate2	:=	Para.rT_Pred_InAirER_Rate2;
		ELSIF Para.rT_Pred_InAirER_Start2 < Para.rT_Pred_InAirER_Start THEN
			rT_Pred_InAirER_Start1	:=	Para.rT_Pred_InAirER_Start2;
			rT_Pred_InAirER_Rate1	:=	Para.rT_Pred_InAirER_Rate2;
			rT_Pred_InAirER_Start2	:=	Para.rT_Pred_InAirER_Start;
			rT_Pred_InAirER_Rate2	:=	Para.rT_Pred_InAirER_Rate;
		ELSIF Para.rT_Pred_InAirER_Start2 = Para.rT_Pred_InAirER_Start THEN
			rT_Pred_InAirER_Start1	:=	Para.rT_Pred_InAirER_Start2;
			rT_Pred_InAirER_Rate1	:=	Para.rT_Pred_InAirER_Rate2;
			rT_Pred_InAirER_Start2	:=	Para.rT_Pred_InAirER_Start;
			rT_Pred_InAirER_Rate2	:=	Para.rT_Pred_InAirER_Rate;
			IF Para.rT_Pred_InAirER_Rate > Para.rT_Pred_InAirER_Rate2 THEN	(* higher reduction is active *)
				rT_Pred_InAirER_Rate1	:=	Para.rT_Pred_InAirER_Rate;
				rT_Pred_InAirER_Rate2	:=	Para.rT_Pred_InAirER_Rate;
			ELSE
				rT_Pred_InAirER_Rate1	:=	Para.rT_Pred_InAirER_Rate2;
				rT_Pred_InAirER_Rate2	:=	Para.rT_Pred_InAirER_Rate2;
			END_IF;
		END_IF;

		IF IN_VE.rT_Ch_T1LP_Avg > rT_Pred_InAirER_Start2 THEN
			rP_Red_T_InAirER_Lim1 := (rT_Pred_InAirER_Start2 - rT_Pred_InAirER_Start1) * rT_Pred_InAirER_Rate1;
			rP_Red_T_InAirER_Lim2 := (IN_VE.rT_Ch_T1LP_Avg    - rT_Pred_InAirER_Start2) * rT_Pred_InAirER_Rate2;
			rP_Red_T_InAirER_Lim  :=  rP_Red_T_InAirER_Lim1  + rP_Red_T_InAirER_Lim2;
		ELSIF IN_VE.rT_Ch_T1LP_Avg > rT_Pred_InAirER_Start1 THEN
			rP_Red_T_InAirER_Lim  := ((IN_VE.rT_Ch_T1LP_Avg   - rT_Pred_InAirER_Start1) * rT_Pred_InAirER_Rate1);
		ELSE
			rP_Red_T_InAirER_Lim  := 0.0;
		END_IF;

		OUT_VE.rP_Red_T_InAirER_Norm := LIMIT(0.5, 1.0 - rP_Red_T_InAirER_Lim, 1.0);
	ELSE
		OUT_VE.rP_Red_T_InAirER_Norm := 1.0;
	END_IF;

END_PROGRAM
```

#### T_InAirER.var
```iecst
VAR
	xGRMAX_T_InAirER_LimHi_Lou : GR_MAXR;
	xGRMAX_T_InAirER_LimHi_Fan : GR_MAXR;
	rT_Pred_InAirER_Start1 : REAL;
	rT_Pred_InAirER_Rate1 : REAL;
	rT_Pred_InAirER_Start2 : REAL;
	rT_Pred_InAirER_Rate2 : REAL;
	rP_Red_T_InAirER_Lim1 : REAL;
	rP_Red_T_InAirER_Lim2 : REAL;
	rP_Red_T_InAirER_Lim : REAL;
END_VAR
```

### Program Logical/Ventilation/T_AirER (IEC, version 3.99.0) - engine room air temperature

#### T_AirERCyclic.st
```iecst
(*******************************************************************************
T_AirER			temperature air engine room

This code is confidential and proprietary to the INNIO Company.
It may not be used in any form, or reproduced in any manner,
without the express written permission of the INNIO Company.
Copyright, INNIO Company, 2019

Customized modifications: -
------------------------

History:
-------
V190	12.08.2004	LH			erstellt
V220	01.03.2007	LH			Erweiterung auf Pt100
 		10.04.2007	LH			Korrektur Messignalüberwachung, Zuweisung für Pt100
V2201	23.07.2007	LH			Messignalüberwachung: UGR -20°C --> -50°C
V3.99.0	14.02.2013	lettenb.	task rtm renamed to T_AirER
V4.14.0 10.12.2024	Nagy		engine room temp high warning added
Instructions for use:
--------------------
Outstandings:
------------
*******************************************************************************)
PROGRAM _CYCLIC

	IF IN_VE.tT_AirER.GoodQual THEN
		rT_AirER := IN_VE.tT_AirER.Ai;			(* standard sensor       engine room temperature *)
	ELSE
		rT_AirER := IN_VE.rT_AirER_Customized;	(* customized preparated engine room temperature *)
	END_IF;

	(* engine room temperature limit warning *)
	xGRMAXR_Hi_Wr(Gw:= Para.rT_AirER_LimWr, Hy:= Para.rT_AirER_HyHi, In:= rT_AirER);
	bT_AirER_Hi_Wr := IN_VE.tPB2MM.bParaSetupOk AND xGRMAXR_Hi_Wr.Q AND Para.bT_AirER_Active;

	(*---------------------------------------------------------------------------*)
	(* engine room temperature limit high *)
	xGRMAXR_Hi(Gw:= Para.rT_AirER_LimHi, Hy:= Para.rT_AirER_HyHi, In:= rT_AirER);
	bT_AirER_Hi := IN_VE.tPB2MM.bParaSetupOk AND xGRMAXR_Hi.Q AND Para.bT_AirER_Active;

	(*---------------------------------------------------------------------------*)
	(* engine room temperature limit 1 (start ventilation(stage 1)) *)
	xGRMAXR_Hi1(Gw:= Para.rT_AirER_LimHi1, Hy:= Para.rT_AirER_HyHi1, In:= rT_AirER);
	bT_AirER_Hi1 := IN_VE.tPB2MM.bParaSetupOk AND xGRMAXR_Hi1.Q AND Para.bT_AirER_Active;

	(*---------------------------------------------------------------------------*)
	(* engine room temperature limit 2 (start ventilation stage 2) *)
	xGRMAXR_Hi2(Gw:= Para.rT_AirER_LimHi2, Hy:= Para.rT_AirER_HyHi2, In:= rT_AirER);
	bT_AirER_Hi2 := IN_VE.tPB2MM.bParaSetupOk AND xGRMAXR_Hi2.Q AND Para.bT_AirER_Active;

	(*---------------------------------------------------------------------------*)
	(* engine room temperature limit 3 (reserve limit value) *)
	xGRMAXR_Hi3(Gw:= Para.rT_AirER_LimHi3, Hy:= Para.rT_AirER_HyHi3, In:= rT_AirER);
	bT_AirER_Hi3 := IN_VE.tPB2MM.bParaSetupOk AND xGRMAXR_Hi3.Q AND Para.bT_AirER_Active;

	(*---------------------------------------------------------------------------*)
	(* engine room temperature limit 4 (start ventilation at engine stop) *)
	xGRMAXR_Hi4(Gw:= Para.rT_AirER_LimHi4, Hy:= Para.rT_AirER_HyHi4, In:= rT_AirER);
	bT_AirER_Hi4  := IN_VE.tPB2MM.bParaSetupOk AND xGRMAXR_Hi4.Q AND Para.bT_AirER_Active;

END_PROGRAM
```

#### T_AirER.var
```iecst
VAR
	xGRMAXR_Hi_Wr : GR_MAXR;
	xGRMAXR_Hi : GR_MAXR;
	xGRMAXR_Hi1 : GR_MAXR;
	xGRMAXR_Hi2 : GR_MAXR;
	xGRMAXR_Hi3 : GR_MAXR;
	xGRMAXR_Hi4 : GR_MAXR;
END_VAR
```

### Program Logical/Ventilation/Ctr_InlLou (IEC, version 4.25.0) - controller engine room temp. with inlet louver(s)

#### Ctr_InlLouCyclic.st
```iecst
(*******************************************************************************
Ctr_InlLou		controller inlet louver(s) to guarantee a constant engine room temperature

This code is confidential and proprietary to the INNIO Company.
It may not be used in any form, or reproduced in any manner,
without the express written permission of the INNIO Company.
Copyright, INNIO Company, 2022

Customized modifications: -
------------------------

History:
-------
V4.03.0	03.08.2015	Stary		created
        19.11.2015  Stary       modified logic for the case "fire-alarm", tCtr_InlLou_In.Y_set_Active, bugfix
		04.12.2015	Stary		writing MM2VIS now with IN_VE.tPos_InlLou1.Ai & IN_VE.tPos_InlLou2.Ai, bugfix
		11.04.2016	stary/lett.	tCtr_InlLou_In.Y_set_Active, tCtr_InlLou_In.Y_set: RTM40 added, bugfix
V4.04.0 17.10.2016  Stary       added RTM40 in ctr-release and external-Y-logic for opening louvers at engine standstill to run ventilation with minimum-speed, bugfix
		26.01.2017	lettenb.	external Y: gasalarm prio before RTM40, bugfix
V4.05.0 20.09.2017	Messner		Active Cooling Program added
V4.11.0	28.01.2022	Perktold	included plant controller upgrade
V4.13.0	05.12.2023	Bacci		Added ventilation demand before starting the ingition selftest and exhaust scavenging
V4.14.0 25.11.2024	Bacci		T6 Start procedure with purge start (2024-219): added ventilation demand before purge cranking cycle during fast start preparation
V4.25.0 26.11.2025	Bacci		Safety Function - Insufficient Ventilation (2024-202): safety plausibility check added

Specification       : PID-controller to ensure a constant room temperature.

Instructions for use: Modify release/X/external Y customized when needed

Outstandings:
------------
(*******************************************************************************)

PROGRAM _CYCLIC

	(* Parameter *)

	Para.tCtr_InlLou.W_set;
	Para.tCtr_InlLou.W_set2;
	Para.tCtr_InlLou.W_min;
	Para.tCtr_InlLou.W_max;
	Para.tCtr_InlLou.dW_up;
	Para.tCtr_InlLou.dW_down;
	Para.tCtr_InlLou.deadband;
	Para.tCtr_InlLou.Y_min;
	Para.tCtr_InlLou.Y_max;
	Para.tCtr_InlLou.dY_max;
	Para.tCtr_InlLou.Y_block;
	Para.tCtr_InlLou.invert;
	Para.tCtr_InlLou.Kp;
	Para.tCtr_InlLou.Tn;
	Para.tCtr_InlLou.Tv;
	Para.tCtr_InlLou.Kp_GainScheduling;
	Para.tCtr_InlLou.Tn_GainScheduling;
	Para.tCtr_InlLou.Tv_GainScheduling;
	Para.tCtr_InlLou.t_min_pulse_down;
	Para.tCtr_InlLou.t_min_pulse_up;
	Para.tCtr_InlLou.t_period_down;
	Para.tCtr_InlLou.t_period_up;

	(* Input variables *)
	tCtr_InlLou_In 				:=	VIS2MM.tCtr_InlLou_In;

	(* Input from module *)
	tCtr_InlLou_In.enable		:=	IN_VE.tPB2MM.bParaSetupOk	(* enable controller *)
							AND		Para.bCtr_InlLou
							AND		(IN_VE.bEng_Aux_Dem_CDR OR IN_VE.bACP_AirER_Dem)
							AND NOT IN_VE.bMsg1052				(* gas pre-alarm *)
							AND NOT IN_VE.bMsg1053      		(* gas alarm *)
							AND NOT IN_VE.bMsg1054      		(* fire alarm *)
							AND NOT MS_LUE    					(* measuring signal failure room temperature --> W3152 *)
							AND NOT RTM40						(* temperature-limit at engine standstill to run ventilation with minimum-speed *)
							AND NOT IN_VE.bInLouDemIgn 			(* ignition self test *)
							AND NOT IN_VE.bInLouDemEX			(* exhaust scavenging *)
							AND NOT IN_VE.bInLouDemAG			(* purge cycle during fast start preparation *)
							AND NOT bERV_SafeCheck_CloseLou		(* safety plausibility check close louvers*)
							AND NOT bERV_SafeCheck_OpenLou;		(* safety plausibility check open louvers*)

	tCtr_InlLou_In.X            :=  rT_AirER;                   (* select X *)

	IF IN_VE.bMsg1052 OR IN_VE.bMsg1053 THEN 					(* external Y at gas pre-alarm/gas alarm/measuring signal failure room temperature *)
		tCtr_InlLou_In.Y_set_Active := TRUE;
		tCtr_InlLou_In.Y_set := 1.0;
	ELSIF IN_VE.bMsg1054 THEN   								(* external Y at fire alarm *)
		tCtr_InlLou_In.Y_set_Active := TRUE;
		tCtr_InlLou_In.Y_set := 0.0;
	ELSIF bERV_SafeCheck_CloseLou THEN
		tCtr_InlLou_In.Y_set_Active := TRUE;
		tCtr_InlLou_In.Y_set := 0.0;
	ELSIF MS_LUE OR RTM40 OR IN_VE.bInLouDemIgn OR IN_VE.bInLouDemEX OR IN_VE.bInLouDemAG OR bERV_SafeCheck_OpenLou THEN
		tCtr_InlLou_In.Y_set_Active := TRUE;
		tCtr_InlLou_In.Y_set := 1.0;
	ELSE
		tCtr_InlLou_In.Y_set_Active := FALSE;
	END_IF;

	IF IN_VE.bACP_AirER_Dem THEN
		tCtr_InlLou_In.W_ext_Active	:= TRUE;
		tCtr_InlLou_In.W_ext		:= Para.rT_ACP_AirER_sp;
	ELSE
		tCtr_InlLou_In.W_ext_Active	:= FALSE;
	END_IF;
	tCtr_InlLou_In.W_set2_Active	:= FALSE;		(*Input to define which internal setpoint will be used TRUE = use the 2nd set point | FALSE use the normal "1st" one*)
	tCtr_InlLou_In.GainScheduling	:= 0.0;			(*Input for Gain Scheduling: 0.0 = use 100% of the Standard PID-Parameters | 1.0 = use 100% of the GainSched. PID Parameters | linear interpolation in between*)
	tCtr_InlLou_In.Y_min_cust		:= -1.0;		(*"customized" Y-Min at the current moment (The existing Y-Min parameter is the global minimum. To have an effect Y_min_cust needs to be > the parameter | -1.0 = function not used*)
	tCtr_InlLou_In.Y_max_cust		:= 1.0;			(*"customized" Y-Max at the current moment (The existing Y-Max parameter is the global maximum. To have an effect Y_max_cust needs to be < the parameter | 1.0 = function not used*)
	tCtr_InlLou_In.Retrigger		:= FALSE;		(*a rising edge on this input signals the controller to retrigger - set W on X and force the Integrator to the current Y*)
	tCtr_InlLou_In.A;								(*optional: feed forward Input*)

	(* Input from Visualization via OPC *)
	tCtr_InlLou_In.Y_man_Active;
	tCtr_InlLou_In.Y_man;
	tCtr_InlLou_In.X_min;
	tCtr_InlLou_In.X_max;
	tCtr_InlLou_In.Tune_quality;
	tCtr_InlLou_In.Tune_PI;
	tCtr_InlLou_In.Tune_PID;
	tCtr_InlLou_In.Tune_start;
	tCtr_InlLou_In.Tune_stop;
	tCtr_InlLou_In.Tune_takeover;

	xCtr_InlLou();

	(* Output variables function block *)
	(* Output to module(s) *)
	OUT_VE.tCtr_InlLou_Set.Ao	:= tCtr_InlLou_Out.Y;	(* analog out *)

	(* Output to Visualization via OPC *)
	MM2VIS.tCtr_InlLou_Out		:= tCtr_InlLou_Out;
	MM2VIS.rPos_InlLou1         := IN_VE.tPos_InlLou1.Ai;
	MM2VIS.rPos_InlLou2			:= IN_VE.tPos_InlLou2.Ai;
	VIS2MM.tCtr_InlLou_In		:= tCtr_InlLou_In;		(* write back to IN_struct for reset: Tune_takeover, X-display, ...!*)

	tCtr_InlLou_Out.Active;
	tCtr_InlLou_Out.Y;
	tCtr_InlLou_Out.W;
	tCtr_InlLou_Out.e;
	tCtr_InlLou_Out.Kp_tune;
	tCtr_InlLou_Out.Tn_tune;
	tCtr_InlLou_Out.Tv_tune;
	tCtr_InlLou_Out.status;
	tCtr_InlLou_Out.Step_down;
	tCtr_InlLou_Out.Step_up;

END_PROGRAM
```

#### Ctr_InlLouInit.st
```iecst
PROGRAM _INIT

	xCtr_InlLou.pParameter 	:= ADR(Para.tCtr_InlLou);
	xCtr_InlLou.pInput 	 	:= ADR(tCtr_InlLou_In);
	xCtr_InlLou.pOutput	 	:= ADR(tCtr_InlLou_Out);

	tCtr_InlLou_In.AlwaysUseYRamp		:= TRUE;	(*If TRUE the Y signal will always limit the change rate via the according parameter | if FALSE the Y signal will jump in case the controller is disabled (blocked or set)*)
	tCtr_InlLou_In.KeepYManAtBlock		:= TRUE;	(*If TRUE the controller will keep the Y-man value constant in case the controller is disabled (blocked or set) | If FALSE the blocked or set value will override the Y-man value*)
	tCtr_InlLou_In.Y_min_cust			:= -1.0;	(*"customized" Y-Min at the current moment (The existing Y-Min parameter is the global minimum. To have an effect Y_min_cust needs to be > the parameter | -1.0 = function not used*)
	tCtr_InlLou_In.Y_max_cust			:=  1.0;	(*"customized" Y-Max at the current moment (The existing Y-Max parameter is the global maximum. To have an effect Y_max_cust needs to be < the parameter | 1.0 = function not used*)
	tCtr_InlLou_In.StepperMode			:= FALSE;	(* TRUE = use PWM-Mode (standard mode until 4.10) | FALSE = use continuous servo drive *)

END_PROGRAM
```

### Program Logical/Ventilation/Ctr_CircLou (IEC, version 4.11.0) - controller engine intake air temp. with circulation louver(s) 

#### Ctr_CircLouCyclic.st
```iecst
(*******************************************************************************
Ctr_CircLou		controller for circulation louver(s) to guarantee a constant engine intake air temperature

This code is confidential and proprietary to the INNIO Company.
It may not be used in any form, or reproduced in any manner,
without the express written permission of the INNIO Company.
Copyright, INNIO Company, 2022

Customized modifications: -
------------------------

History:
-------
V4.03.0		03.08.2015		Stary		created
			04.12.2015		Stary		bugfix: line92,93
                                        		writing MM2VIS now with IN_VE.tPos_CircLou1.Ai & IN_VE.tPos_CircLou2.Ai
V4.11.0		28.01.2022		Perktold	included plant controller upgrade

Specification       : PID-controller to ensure a constant engine intake air temperature

Instructions for use: Modify release/X/external Y customized when needed

Outstandings:
------------
(*******************************************************************************)

PROGRAM _CYCLIC

	(* Parameter *)

	Para.tCtr_CircLou.W_set;
	Para.tCtr_CircLou.W_set2;
	Para.tCtr_CircLou.W_min;
	Para.tCtr_CircLou.W_max;
	Para.tCtr_CircLou.dW_up;
	Para.tCtr_CircLou.dW_down;
	Para.tCtr_CircLou.deadband;
	Para.tCtr_CircLou.Y_min;
	Para.tCtr_CircLou.Y_max;
	Para.tCtr_CircLou.dY_max;
	Para.tCtr_CircLou.Y_block;
	Para.tCtr_CircLou.invert;
	Para.tCtr_CircLou.Kp;
	Para.tCtr_CircLou.Tn;
	Para.tCtr_CircLou.Tv;
	Para.tCtr_CircLou.Kp_GainScheduling;
	Para.tCtr_CircLou.Tn_GainScheduling;
	Para.tCtr_CircLou.Tv_GainScheduling;
	Para.tCtr_CircLou.t_min_pulse_down;
	Para.tCtr_CircLou.t_min_pulse_up;
	Para.tCtr_CircLou.t_period_down;
	Para.tCtr_CircLou.t_period_up;

	(* Input variables *)
	tCtr_CircLou_In 				:= VIS2MM.tCtr_CircLou_In;

	(* Input from module *)

	xGR_MINR_CircLou(In := IN_VE.rT_Ch_T1LP_Avg, Gw := Para.rT_InAirER_Rel_CircOp, Hy := Para.rT_InAirER_Rel_CircOp_Hy);	(* release of circulation operation regarding engine air intake temp. *)
    bRel_CircOp := xGR_MINR_CircLou.Q;

	tCtr_CircLou_In.enable		:=	IN_VE.tPB2MM.bParaSetupOk		(* enable controller *)
										AND		Para.bCtr_CircLou
										AND     bRel_CircOp
										AND NOT IN_VE.bMsg1052		(* gas pre-alarm *)
										AND NOT IN_VE.bMsg1053      (* gas alarm *)
										AND NOT IN_VE.bMsg1054;     (* fire alarm *)

	tCtr_CircLou_In.X            :=  IN_VE.rT_Ch_T1LP_Avg;          (* select X *)

	tCtr_CircLou_In.Y_set_Active := IN_VE.bMsg1052 OR IN_VE.bMsg1053 OR IN_VE.bMsg1054 OR NOT bRel_CircOp;	(* external Y at gas pre-alarm/gas alarm/fire-alarm/no release circ. OP *)
	tCtr_CircLou_In.Y_set 			:= 0.0;
	tCtr_CircLou_In.W_set2_Active	:= FALSE;		(*Input to define which internal setpoint will be used TRUE = use the 2nd set point | FALSE use the normal "1st" one*)
	tCtr_CircLou_In.GainScheduling	:= 0.0;			(*Input for Gain Scheduling: 0.0 = use 100% of the Standard PID-Parameters | 1.0 = use 100% of the GainSched. PID Parameters | linear interpolation in between*)
	tCtr_CircLou_In.Y_min_cust		:= -1.0;		(*"customized" Y-Min at the current moment (The existing Y-Min parameter is the global minimum. To have an effect Y_min_cust needs to be > the parameter | -1.0 = function not used*)
	tCtr_CircLou_In.Y_max_cust		:= 1.0;			(*"customized" Y-Max at the current moment (The existing Y-Max parameter is the global maximum. To have an effect Y_max_cust needs to be < the parameter | 1.0 = function not used*)
	tCtr_CircLou_In.Retrigger		:= FALSE;		(*a rising edge on this input signals the controller to retrigger - set W on X and force the Integrator to the current Y*)
	tCtr_CircLou_In.A;								(*optional: feed forward Input*)

	(* Input from Visualization via OPC *)
	tCtr_CircLou_In.Y_man_Active;
	tCtr_CircLou_In.Y_man;
	tCtr_CircLou_In.X_min;
	tCtr_CircLou_In.X_max;
	tCtr_CircLou_In.Tune_quality;
	tCtr_CircLou_In.Tune_PI;
	tCtr_CircLou_In.Tune_PID;
	tCtr_CircLou_In.Tune_start;
	tCtr_CircLou_In.Tune_stop;
	tCtr_CircLou_In.Tune_takeover;

	xCtr_CircLou();

	(* Output variables function block *)
	(* Output to module(s) *)
	OUT_VE.tCtr_CircLou_Set.Ao	:= tCtr_CircLou_Out.Y;	(* analog out *)

	(* Output to Visualization via OPC *)
	MM2VIS.tCtr_CircLou_Out		:= tCtr_CircLou_Out;
	MM2VIS.rPos_CircLou1            := IN_VE.tPos_CircLou1.Ai;
	MM2VIS.rPos_CircLou2		:= IN_VE.tPos_CircLou2.Ai;
	VIS2MM.tCtr_CircLou_In		:= tCtr_CircLou_In;		(* write back to IN_struct for reset: Tune_takeover, X-display, ...!*)

	tCtr_CircLou_Out.Active;
	tCtr_CircLou_Out.Y;
	tCtr_CircLou_Out.W;
	tCtr_CircLou_Out.e;
	tCtr_CircLou_Out.Kp_tune;
	tCtr_CircLou_Out.Tn_tune;
	tCtr_CircLou_Out.Tv_tune;
	tCtr_CircLou_Out.status;
	tCtr_CircLou_Out.Step_down;
	tCtr_CircLou_Out.Step_up;

END_PROGRAM
```

#### Ctr_CircLouInit.st
```iecst
PROGRAM _INIT

	xCtr_CircLou.pParameter  := ADR(Para.tCtr_CircLou);
	xCtr_CircLou.pInput 	 := ADR(tCtr_CircLou_In);
	xCtr_CircLou.pOutput	 := ADR(tCtr_CircLou_Out);

	tCtr_CircLou_In.AlwaysUseYRamp		:= TRUE;	(*If TRUE the Y signal will always limit the change rate via the according parameter | if FALSE the Y signal will jump in case the controller is disabled (blocked or set)*)
	tCtr_CircLou_In.KeepYManAtBlock		:= TRUE;	(*If TRUE the controller will keep the Y-man value constant in case the controller is disabled (blocked or set) | If FALSE the blocked or set value will override the Y-man value*)
	tCtr_CircLou_In.Y_min_cust			:= -1.0;	(*"customized" Y-Min at the current moment (The existing Y-Min parameter is the global minimum. To have an effect Y_min_cust needs to be > the parameter | -1.0 = function not used*)
	tCtr_CircLou_In.Y_max_cust			:=  1.0;	(*"customized" Y-Max at the current moment (The existing Y-Max parameter is the global maximum. To have an effect Y_max_cust needs to be < the parameter | 1.0 = function not used*)
	tCtr_CircLou_In.StepperMode			:= FALSE;	(* TRUE = use PWM-Mode (standard mode until 4.10) | FALSE = use continuous servo drive *)

END_PROGRAM
```

#### Ctr_CircLou.var
```iecst
VAR
	bRel_CircOp : BOOL; (*air circulating operation released*)
	xGR_MINR_CircLou : GR_MINR := (0); (*maximum engine intake air temperature for release circulating operation (STM)*)
END_VAR
```

### Program Logical/Ventilation/Ctr_OutLRT (IEC, version 4.25.0) - controller engine room temp. with outlet louver(s)

#### Ctr_OutLRTCyclic.st
```iecst
(*******************************************************************************
Ctr_OutlLou_RT		controller for outlet louver(s) to guarantee a constant engine room temperature

This code is confidential and proprietary to the INNIO Company.
It may not be used in any form, or reproduced in any manner,
without the express written permission of the INNIO Company.
Copyright, INNIO Company, 2022

Customized modifications: -
------------------------

History:
-------
V4.03.0	24.09.2015	Stary		created
  		19.11.2015  Stary       modified logic FOR the CASE "fire-alarm", tCtr_OutlLou_RT_In.Y_set_Active, bugfix
		04.12.2015	Stary		writing MM2VIS now with IN_VE.tPos_OutlLou1.Ai & IN_VE.tPos_OutlLou2.Ai, bugfix
		11.04.2016	stary/lett.	tCtr_OutlLou_RT_In.Y_set_Active, tCtr_OutlLou_RT_In.Y_set: RTM40 added, bugfix
V4.04.0 17.10.2016  Stary       added RTM40 in ctr-release and external-Y-logic for opening louvers at engine standstill to run ventilation with minimum-speed, bugfix
		26.01.2017	lettenb.	external Y: gasalarm prio before RTM40, bugfix
		03.07.2017	lettenb.	tCtr_OutlLou_In.Y_set -> tCtr_OutlLou_RT_In.Y_set removed, bugfix
V4.11.0	28.01.2022	Perktold	included plant controller upgrade
V4.25.0 26.11.2025	Bacci		Safety Function - Insufficient Ventilation (2024-202): safety plausibility check added

Specification       : PID-controller for outlet louver(s) to ensure a constant room temperature

Instructions for use: Modify release/X/external Y customized when needed

Outstandings:
------------
(*******************************************************************************)

PROGRAM _CYCLIC

	(* Parameter *)

	Para.tCtr_OutlLou_RT.W_set;
	Para.tCtr_OutlLou_RT.W_set2;
	Para.tCtr_OutlLou_RT.W_min;
	Para.tCtr_OutlLou_RT.W_max;
	Para.tCtr_OutlLou_RT.dW_up;
	Para.tCtr_OutlLou_RT.dW_down;
	Para.tCtr_OutlLou_RT.deadband;
	Para.tCtr_OutlLou_RT.Y_min;
	Para.tCtr_OutlLou_RT.Y_max;
	Para.tCtr_OutlLou_RT.dY_max;
	Para.tCtr_OutlLou_RT.Y_block;
	Para.tCtr_OutlLou_RT.invert;
	Para.tCtr_OutlLou_RT.Kp;
	Para.tCtr_OutlLou_RT.Tn;
	Para.tCtr_OutlLou_RT.Tv;
	Para.tCtr_OutlLou_RT.Kp_GainScheduling;
	Para.tCtr_OutlLou_RT.Tn_GainScheduling;
	Para.tCtr_OutlLou_RT.Tv_GainScheduling;
	Para.tCtr_OutlLou_RT.t_min_pulse_down;
	Para.tCtr_OutlLou_RT.t_min_pulse_up;
	Para.tCtr_OutlLou_RT.t_period_down;
	Para.tCtr_OutlLou_RT.t_period_up;

	(* Input variables *)
	tCtr_OutlLou_RT_In				:= VIS2MM.tCtr_OutlLou_RT_In;

	(* Input from module *)
	tCtr_OutlLou_RT_In.enable		:=	IN_VE.tPB2MM.bParaSetupOk		(* enable controller *)
									AND		Para.bCtr_OutlLou_RT
									AND     IN_VE.bEng_Aux_Dem_CDR
									AND NOT IN_VE.bMsg1052				(* gas pre-alarm *)
									AND NOT IN_VE.bMsg1053      		(* gas alarm *)
									AND NOT IN_VE.bMsg1054      		(* fire alarm *)
									AND NOT MS_LUE    					(* measuring signal failure room temperature *)
									AND NOT RTM40						(* temperature-limit at engine standstill to run ventilation with minimum-speed *)
									AND NOT bERV_SafeCheck_CloseLou		(* safety plausibility check close louvers*)
									AND NOT bERV_SafeCheck_OpenLou;		(* safety plausibility check open louvers*)

	tCtr_OutlLou_RT_In.X			:=	rT_AirER;

	IF IN_VE.bMsg1052 OR IN_VE.bMsg1053 THEN							(* external Y --> totally open the louver(s) at gas-pre-alarm/gas-alarm *)
		tCtr_OutlLou_RT_In.Y_set_Active := TRUE;
		tCtr_OutlLou_RT_In.Y_set := 1.0;
	ELSIF IN_VE.bMsg1054 THEN 											(* external Y --> totally close the louver(s) at fire-alarm *)
		tCtr_OutlLou_RT_In.Y_set_Active := TRUE;
		tCtr_OutlLou_RT_In.Y_set := 0.0;
	ELSIF bERV_SafeCheck_CloseLou THEN
		tCtr_InlLou_In.Y_set_Active := TRUE;
		tCtr_InlLou_In.Y_set := 0.0;
	ELSIF MS_LUE OR RTM40 OR bERV_SafeCheck_OpenLou THEN
		tCtr_OutlLou_RT_In.Y_set_Active := TRUE;
		tCtr_OutlLou_RT_In.Y_set := 1.0;
	ELSE
		tCtr_OutlLou_RT_In.Y_set_Active := FALSE;
	END_IF;
	tCtr_OutlLou_RT_In.W_set2_Active	:= FALSE;		(*Input to define which internal setpoint will be used TRUE = use the 2nd set point | FALSE use the normal "1st" one*)
	tCtr_OutlLou_RT_In.GainScheduling	:= 0.0;			(*Input for Gain Scheduling: 0.0 = use 100% of the Standard PID-Parameters | 1.0 = use 100% of the GainSched. PID Parameters | linear interpolation in between*)
	tCtr_OutlLou_RT_In.Y_min_cust		:= -1.0;		(*"customized" Y-Min at the current moment (The existing Y-Min parameter is the global minimum. To have an effect Y_min_cust needs to be > the parameter | -1.0 = function not used*)
	tCtr_OutlLou_RT_In.Y_max_cust		:= 1.0;			(*"customized" Y-Max at the current moment (The existing Y-Max parameter is the global maximum. To have an effect Y_max_cust needs to be < the parameter | 1.0 = function not used*)
	tCtr_OutlLou_RT_In.Retrigger		:= FALSE;		(*a rising edge on this input signals the controller to retrigger - set W on X and force the Integrator to the current Y*)
	tCtr_OutlLou_RT_In.A;								(*optional: feed forward Input*)

	(* Input from Visualization via OPC *)
	tCtr_OutlLou_RT_In.Y_man_Active;
	tCtr_OutlLou_RT_In.Y_man;
	tCtr_OutlLou_RT_In.X_min;
	tCtr_OutlLou_RT_In.X_max;
	tCtr_OutlLou_RT_In.Tune_quality;
	tCtr_OutlLou_RT_In.Tune_PI;
	tCtr_OutlLou_RT_In.Tune_PID;
	tCtr_OutlLou_RT_In.Tune_start;
	tCtr_OutlLou_RT_In.Tune_stop;
	tCtr_OutlLou_RT_In.Tune_takeover;

	xCtr_OutlLou_RT();

	(* Output variables function block *)
	(* Output to module(s) *)
	OUT_VE.tCtr_OutlLou_RT_Set.Ao	:= tCtr_OutlLou_RT_Out.Y;	(* analog out *)

	(* Output to Visualization via OPC *)
	MM2VIS.tCtr_OutlLou_RT_Out	:= tCtr_OutlLou_RT_Out;
	MM2VIS.rPos_OutlLou1        := IN_VE.tPos_OutlLou1.Ai;
	MM2VIS.rPos_OutlLou2        := IN_VE.tPos_OutlLou2.Ai;
	VIS2MM.tCtr_OutlLou_RT_In	:= tCtr_OutlLou_RT_In;		(* write back to IN_struct for reset: Tune_takeover, X-display, ...!*)

	tCtr_OutlLou_RT_Out.Active;
	tCtr_OutlLou_RT_Out.Y;
	tCtr_OutlLou_RT_Out.W;
	tCtr_OutlLou_RT_Out.e;
	tCtr_OutlLou_RT_Out.Kp_tune;
	tCtr_OutlLou_RT_Out.Tn_tune;
	tCtr_OutlLou_RT_Out.Tv_tune;
	tCtr_OutlLou_RT_Out.status;
	tCtr_OutlLou_RT_Out.Step_down;
	tCtr_OutlLou_RT_Out.Step_up;

END_PROGRAM
```

#### Ctr_OutLRTInit.st
```iecst
PROGRAM _INIT

	xCtr_OutlLou_RT.pParameter 	:= ADR(Para.tCtr_OutlLou_RT); (*STM 2*)
	xCtr_OutlLou_RT.pInput 	 	:= ADR(tCtr_OutlLou_RT_In); (*STM 2*)
	xCtr_OutlLou_RT.pOutput	 	:= ADR(tCtr_OutlLou_RT_Out); (*STM 2*)

	tCtr_OutlLou_RT_In.AlwaysUseYRamp		:= TRUE;	(*If TRUE the Y signal will always limit the change rate via the according parameter | if FALSE the Y signal will jump in case the controller is disabled (blocked or set)*)
	tCtr_OutlLou_RT_In.KeepYManAtBlock		:= TRUE;	(*If TRUE the controller will keep the Y-man value constant in case the controller is disabled (blocked or set) | If FALSE the blocked or set value will override the Y-man value*)
	tCtr_OutlLou_RT_In.Y_min_cust			:= -1.0;	(*"customized" Y-Min at the current moment (The existing Y-Min parameter is the global minimum. To have an effect Y_min_cust needs to be > the parameter | -1.0 = function not used*)
	tCtr_OutlLou_RT_In.Y_max_cust			:=  1.0;	(*"customized" Y-Max at the current moment (The existing Y-Max parameter is the global maximum. To have an effect Y_max_cust needs to be < the parameter | 1.0 = function not used*)
	tCtr_OutlLou_RT_In.StepperMode			:= FALSE;	(* TRUE = use PWM-Mode (standard mode until 4.10) | FALSE = use continuous servo drive *)

END_PROGRAM
```

### Program Logical/Ventilation/Ctr_OutLRDP (IEC, version 4.25.0) - controller engine room differential pressure with outlet louver(s)

#### Ctr_OutLRDPCyclic.st
```iecst
(*******************************************************************************
Ctr_OutlLou_RDP		controller for outlet louver(s) to guarantee a constant engine room differential pressure

This code is confidential and proprietary to the INNIO Company.
It may not be used in any form, or reproduced in any manner,
without the express written permission of the INNIO Company.
Copyright, INNIO Company, 2022

Customized modifications: -
------------------------

History:
-------
V4.03.0		24.09.2015		Stary		created
            19.11.2015      Stary       bugfix: line 71
												modified logic FOR the CASE "fire-alarm"
												line 75
												tCtr_OutlLou_RDP_In.Y_set_Active was never resetted
			04.12.2015		Stary		bugfix: line104,105
                                        		writing MM2VIS now with IN_VE.tPos_OutlLou1.Ai & IN_VE.tPos_OutlLou2.Ai
V4.04.0		06.10.2016		Stary       line76: shortened the ELSIF logic cause bMsg1052+bMsg1053+bMsg2705 NOT needed here
V4.04.0		17.10.2016  	Stary       added RTM40 in ctr-release AND external-Y-logic FOR opening louvers at engine standstill TO run ventilation with minimum-speed, bugfix
			15.02.2017	    Stary		external Y: gasalarm prio before RTM40, bugfix
V4.07.0		04.03.2019		lettenb.	IN_VE.bMsg2705 -> OUT_VE.bMsg2705, mapping cleanup
V4.11.0		28.01.2022		Perktold	included plant controller upgrade
V4.25.0		26.11.2025	Bacci		Safety Function - Insufficient Ventilation (2024-202): safety plausibility check added

Specification       : PID-controller for outlet louver(s) to ensure a constant room temperature

Instructions for use: Modify release/X/external Y customized when needed

Outstandings:
------------
(*******************************************************************************)

PROGRAM _CYCLIC

	(* Parameter *)

	Para.tCtr_OutlLou_RDP.W_set;
	Para.tCtr_OutlLou_RDP.W_set2;
	Para.tCtr_OutlLou_RDP.W_min;
	Para.tCtr_OutlLou_RDP.W_max;
	Para.tCtr_OutlLou_RDP.dW_up;
	Para.tCtr_OutlLou_RDP.dW_down;
	Para.tCtr_OutlLou_RDP.deadband;
	Para.tCtr_OutlLou_RDP.Y_min;
	Para.tCtr_OutlLou_RDP.Y_max;
	Para.tCtr_OutlLou_RDP.dY_max;
	Para.tCtr_OutlLou_RDP.Y_block;
	Para.tCtr_OutlLou_RDP.invert;
	Para.tCtr_OutlLou_RDP.Kp;
	Para.tCtr_OutlLou_RDP.Tn;
	Para.tCtr_OutlLou_RDP.Tv;
	Para.tCtr_OutlLou_RDP.Kp_GainScheduling;
	Para.tCtr_OutlLou_RDP.Tn_GainScheduling;
	Para.tCtr_OutlLou_RDP.Tv_GainScheduling;
	Para.tCtr_OutlLou_RDP.t_min_pulse_down;
	Para.tCtr_OutlLou_RDP.t_min_pulse_up;
	Para.tCtr_OutlLou_RDP.t_period_down;
	Para.tCtr_OutlLou_RDP.t_period_up;

	(* Input variables *)
	tCtr_OutlLou_RDP_In				:= VIS2MM.tCtr_OutlLou_RDP_In;

	(* Input from module *)
	tCtr_OutlLou_RDP_In.enable		:=	IN_VE.tPB2MM.bParaSetupOk		(* enable controller *)
									AND		Para.bCtr_OutlLou_RDP
									AND     IN_VE.bEng_Aux_Dem_CDR
									AND NOT IN_VE.bMsg1052				(* gas pre-alarm *)
									AND NOT IN_VE.bMsg1053      		(* gas alarm *)
									AND NOT IN_VE.bMsg1054      		(* fire alarm *)
									AND NOT OUT_VE.bMsg2705    			(* measuring signal failure room differential pressure *)
									AND NOT RTM40						(* temperature-limit at engine standstill to run ventilation with minimum-speed *)
									AND NOT bERV_SafeCheck_CloseLou		(* safety plausibility check close louvers*)
									AND NOT bERV_SafeCheck_OpenLou;		(* safety plausibility check open louvers*)

	tCtr_OutlLou_RDP_In.X			:= IN_VE.tPrDiff_ER.Ai;

	IF IN_VE.bMsg1052 OR IN_VE.bMsg1053 OR (OUT_VE.bMsg2705 AND NOT bERV_SafeCheck_CloseLou) THEN	(* external Y --> totally open the louver(s) at gas-pre-alarm/gas-alarm *)
		tCtr_OutlLou_RDP_In.Y_set_Active := TRUE;
		tCtr_OutlLou_RDP_In.Y_set := 1.0;
	ELSIF IN_VE.bMsg1054 THEN									(* external Y --> totally close the louver(s) at fire-alarm *)
		tCtr_OutlLou_RDP_In.Y_set_Active := TRUE;
		tCtr_OutlLou_RDP_In.Y_set := 0.0;
	ELSIF bERV_SafeCheck_CloseLou THEN
		tCtr_InlLou_In.Y_set_Active := TRUE;
		tCtr_InlLou_In.Y_set := 0.0;
	ELSIF RTM40 OR bERV_SafeCheck_OpenLou THEN
		tCtr_OutlLou_RDP_In.Y_set_Active := TRUE;
		tCtr_OutlLou_RDP_In.Y_set := 1.0;
	ELSE
		tCtr_OutlLou_RDP_In.Y_set_Active := FALSE;
	END_IF;
	tCtr_OutlLou_RDP_In.W_set2_Active	:= FALSE;		(*Input to define which internal setpoint will be used TRUE = use the 2nd set point | FALSE use the normal "1st" one*)
	tCtr_OutlLou_RDP_In.GainScheduling	:= 0.0;			(*Input for Gain Scheduling: 0.0 = use 100% of the Standard PID-Parameters | 1.0 = use 100% of the GainSched. PID Parameters | linear interpolation in between*)
	tCtr_OutlLou_RDP_In.Y_min_cust		:= -1.0;		(*"customized" Y-Min at the current moment (The existing Y-Min parameter is the global minimum. To have an effect Y_min_cust needs to be > the parameter | -1.0 = function not used*)
	tCtr_OutlLou_RDP_In.Y_max_cust		:= 1.0;			(*"customized" Y-Max at the current moment (The existing Y-Max parameter is the global maximum. To have an effect Y_max_cust needs to be < the parameter | 1.0 = function not used*)
	tCtr_OutlLou_RDP_In.Retrigger		:= FALSE;		(*a rising edge on this input signals the controller to retrigger - set W on X and force the Integrator to the current Y*)
	tCtr_OutlLou_RDP_In.A;								(*optional: feed forward Input*)

	(* Input from Visualization via OPC *)
	tCtr_OutlLou_RDP_In.Y_man_Active;
	tCtr_OutlLou_RDP_In.Y_man;
	tCtr_OutlLou_RDP_In.X_min;
	tCtr_OutlLou_RDP_In.X_max;
	tCtr_OutlLou_RDP_In.Tune_quality;
	tCtr_OutlLou_RDP_In.Tune_PI;
	tCtr_OutlLou_RDP_In.Tune_PID;
	tCtr_OutlLou_RDP_In.Tune_start;
	tCtr_OutlLou_RDP_In.Tune_stop;
	tCtr_OutlLou_RDP_In.Tune_takeover;

	xCtr_OutlLou_RDP();

	(* Output variables function block *)
	(* Output to module(s) *)
	OUT_VE.tCtr_OutlLou_RDP_Set.Ao	:= tCtr_OutlLou_RDP_Out.Y;	(* analog out *)

	(* Output to Visualization via OPC *)
	MM2VIS.tCtr_OutlLou_RDP_Out	:= tCtr_OutlLou_RDP_Out;
	MM2VIS.rPos_OutlLou1        := IN_VE.tPos_OutlLou1.Ai;
	MM2VIS.rPos_OutlLou2        := IN_VE.tPos_OutlLou2.Ai;
	VIS2MM.tCtr_OutlLou_RDP_In	:= tCtr_OutlLou_RDP_In;		(* write back to IN_struct for reset: Tune_takeover, X-display, ...!*)

	tCtr_OutlLou_RDP_Out.Active;
	tCtr_OutlLou_RDP_Out.Y;
	tCtr_OutlLou_RDP_Out.W;
	tCtr_OutlLou_RDP_Out.e;
	tCtr_OutlLou_RDP_Out.Kp_tune;
	tCtr_OutlLou_RDP_Out.Tn_tune;
	tCtr_OutlLou_RDP_Out.Tv_tune;
	tCtr_OutlLou_RDP_Out.status;
	tCtr_OutlLou_RDP_Out.Step_down;
	tCtr_OutlLou_RDP_Out.Step_up;

END_PROGRAM
```

#### Ctr_OutLRDPnit.st
```iecst
PROGRAM _INIT

	xCtr_OutlLou_RDP.pParameter 	:= ADR(Para.tCtr_OutlLou_RDP); (*STM 2*)
	xCtr_OutlLou_RDP.pInput 	 	:= ADR(tCtr_OutlLou_RDP_In); (*STM 2*)
	xCtr_OutlLou_RDP.pOutput	 	:= ADR(tCtr_OutlLou_RDP_Out); (*STM 2*)

	tCtr_OutlLou_RDP_In.AlwaysUseYRamp		:= TRUE;	(*If TRUE the Y signal will always limit the change rate via the according parameter | if FALSE the Y signal will jump in case the controller is disabled (blocked or set)*)
	tCtr_OutlLou_RDP_In.KeepYManAtBlock		:= TRUE;	(*If TRUE the controller will keep the Y-man value constant in case the controller is disabled (blocked or set) | If FALSE the blocked or set value will override the Y-man value*)
	tCtr_OutlLou_RDP_In.Y_min_cust			:= -1.0;	(*"customized" Y-Min at the current moment (The existing Y-Min parameter is the global minimum. To have an effect Y_min_cust needs to be > the parameter | -1.0 = function not used*)
	tCtr_OutlLou_RDP_In.Y_max_cust			:=  1.0;	(*"customized" Y-Max at the current moment (The existing Y-Max parameter is the global maximum. To have an effect Y_max_cust needs to be < the parameter | 1.0 = function not used*)
	tCtr_OutlLou_RDP_In.StepperMode			:= FALSE;	(* TRUE = use PWM-Mode (standard mode until 4.10) | FALSE = use continuous servo drive *)

END_PROGRAM
```

### Program Logical/Ventilation/Ctr_OutVRT (IEC, version 4.11.0) - controller engine room temperature with outlet ventilation fan(s)

#### Ctr_OutVRTCyclic.st
```iecst
(*******************************************************************************
Ctr_OutlVentRT		controller engine room temperature with outlet ventilation fan(s)

This code is confidential and proprietary to the INNIO Company.
It may not be used in any form, or reproduced in any manner,
without the express written permission of the INNIO Company.
Copyright, INNIO Company, 2022

Customized modifications: -
------------------------

History:
-------
V4.04.0		04.10.2016	Stary			created
V4.11.0		28.01.2022	Perktold		included plant controller upgrade

Specification       : PID-controller for outlet ventilation fan(s) to ensure a constant room temperature

Instructions for use: Modify release/X/external Y customized when needed
--------------------

Outstandings:
------------
(*******************************************************************************)

PROGRAM _CYCLIC

	(* Parameter *)
	Para.tCtr_OutlVE_RT.W_set;
	Para.tCtr_OutlVE_RT.W_set2;
	Para.tCtr_OutlVE_RT.W_min;
	Para.tCtr_OutlVE_RT.W_max;
	Para.tCtr_OutlVE_RT.dW_up;
	Para.tCtr_OutlVE_RT.dW_down;
	Para.tCtr_OutlVE_RT.deadband;
	Para.tCtr_OutlVE_RT.Y_min;
	Para.tCtr_OutlVE_RT.Y_max;
	Para.tCtr_OutlVE_RT.dY_max;
	Para.tCtr_OutlVE_RT.Y_block;
	Para.tCtr_OutlVE_RT.invert;
	Para.tCtr_OutlVE_RT.Kp;
	Para.tCtr_OutlVE_RT.Tn;
	Para.tCtr_OutlVE_RT.Tv;
	Para.tCtr_OutlVE_RT.Kp_GainScheduling;
	Para.tCtr_OutlVE_RT.Tn_GainScheduling;
	Para.tCtr_OutlVE_RT.Tv_GainScheduling;
	Para.tCtr_OutlVE_RT.t_min_pulse_down;
	Para.tCtr_OutlVE_RT.t_min_pulse_up;
	Para.tCtr_OutlVE_RT.t_period_down;
	Para.tCtr_OutlVE_RT.t_period_up;

	(* Input variables *)
	tCtr_OutlVE_RT_In	 		:= VIS2MM.tCtr_OutlVE_RT_In;

	(* Input from module *)
	tCtr_OutlVE_RT_In.enable	:=	IN_VE.tPB2MM.bParaSetupOk		(* enable controller *)
							AND	    Para.bCtr_OutlVE_RT
							AND     OUT_VE.tRel_ER_FC.Do
							AND	    RTM25
							AND     OUT_VE.tRel_ER_Fan.Do
							AND NOT MS_LUE
							AND NOT bCtrER_YFix;

	tCtr_OutlVE_RT_In.W_ext_Active	:= tCtr_OutlVE_RT_In.W_ext_Active OR TRUE;	(* select external W *) //from visu

	IF IN_VE.bEng_Aux_Dem_CDR THEN
		tCtr_OutlVE_RT_In.W_ext :=	 Para.rT_CtrER_WexRun;					(* external W --> same parameter as for inlet fans *)
	ELSE
		tCtr_OutlVE_RT_In.W_ext :=	 Para.rT_CtrER_WexStop;					(* external W --> same parameter as for inlet fans *)
	END_IF;
	tCtr_OutlVE_RT_In.W_set2_Active		:= FALSE;		(*Input to define which internal setpoint will be used TRUE = use the 2nd set point | FALSE use the normal "1st" one*)
	tCtr_OutlVE_RT_In.GainScheduling	:= 0.0;			(*Input for Gain Scheduling: 0.0 = use 100% of the Standard PID-Parameters | 1.0 = use 100% of the GainSched. PID Parameters | linear interpolation in between*)
	tCtr_OutlVE_RT_In.Y_min_cust		:= -1.0;		(*"customized" Y-Min at the current moment (The existing Y-Min parameter is the global minimum. To have an effect Y_min_cust needs to be > the parameter | -1.0 = function not used*)
	tCtr_OutlVE_RT_In.Y_max_cust		:= 1.0;			(*"customized" Y-Max at the current moment (The existing Y-Max parameter is the global maximum. To have an effect Y_max_cust needs to be < the parameter | 1.0 = function not used*)
	tCtr_OutlVE_RT_In.Retrigger			:= FALSE;		(*a rising edge on this input signals the controller to retrigger - set W on X and force the Integrator to the current Y*)
	tCtr_OutlVE_RT_In.A;								(*optional: feed forward Input*)

	IF bCtrER_YFix THEN
		tCtr_OutlVE_RT_In.Y_set_Active  := bCtrER_YFix; 	 				(* select external Y *)
		tCtr_OutlVE_RT_In.Y_set         := 1.0;
	ELSIF  (NOT tCtr_OutlVE_RT_In.enable
		AND OUT_VE.tRel_ER_FC.Do
		AND IN_VE.tManAuxCtr.bER_OutlV_FC_Set) THEN	(* Manual operating auxiliaries control - Handbedienebene *)
		tCtr_OutlVE_RT_In.Y_set_Active  := TRUE;
		tCtr_OutlVE_RT_In.Y_set         := IN_VE.tManAuxCtr.rER_OutlV_FC_Set;
	ELSE
		tCtr_OutlVE_RT_In.Y_set_Active  := FALSE;
	END_IF;

	tCtr_OutlVE_RT_In.X := rT_AirER;			(* select X *)

	(* Input from Visualization via OPC *)
	tCtr_OutlVE_RT_In.Y_man_Active;
	tCtr_OutlVE_RT_In.Y_man;
	tCtr_OutlVE_RT_In.X_min;
	tCtr_OutlVE_RT_In.X_max;
	tCtr_OutlVE_RT_In.Tune_quality;
	tCtr_OutlVE_RT_In.Tune_PI;
	tCtr_OutlVE_RT_In.Tune_PID;
	tCtr_OutlVE_RT_In.Tune_start;
	tCtr_OutlVE_RT_In.Tune_stop;
	tCtr_OutlVE_RT_In.Tune_takeover;

	xCtr_OutlVE_RT();

	(* Output variables function block *)
	(* Output to module(s) *)
	OUT_VE.tCtr_OutlVE_RT_Set.Ao 	:= tCtr_OutlVE_RT_Out.Y;	(* analog out *)

	(* Output to Visualization via OPC *)
	MM2VIS.tCtr_OutlVE_RT_Out		:= tCtr_OutlVE_RT_Out;
	VIS2MM.tCtr_OutlVE_RT_In		:= tCtr_OutlVE_RT_In;		(* write back to IN_struct for reset: Tune_takeover, X-display, ...!*)

	tCtr_OutlVE_RT_Out.Active;
	tCtr_OutlVE_RT_Out.Y;
	tCtr_OutlVE_RT_Out.W;
	tCtr_OutlVE_RT_Out.e;
	tCtr_OutlVE_RT_Out.Kp_tune;
	tCtr_OutlVE_RT_Out.Tn_tune;
	tCtr_OutlVE_RT_Out.Tv_tune;
	tCtr_OutlVE_RT_Out.status;
	tCtr_OutlVE_RT_Out.Step_down;
	tCtr_OutlVE_RT_Out.Step_up;

END_PROGRAM
```

#### Ctr_OutVRTInit.st
```iecst
PROGRAM _INIT

	xCtr_OutlVE_RT.pParameter 	:= ADR(Para.tCtr_OutlVE_RT);
	xCtr_OutlVE_RT.pInput 	 	:= ADR(tCtr_OutlVE_RT_In);
	xCtr_OutlVE_RT.pOutput	 	:= ADR(tCtr_OutlVE_RT_Out);

	tCtr_OutlVE_RT_In.AlwaysUseYRamp		:= TRUE;	(*If TRUE the Y signal will always limit the change rate via the according parameter | if FALSE the Y signal will jump in case the controller is disabled (blocked or set)*)
	tCtr_OutlVE_RT_In.KeepYManAtBlock		:= TRUE;	(*If TRUE the controller will keep the Y-man value constant in case the controller is disabled (blocked or set) | If FALSE the blocked or set value will override the Y-man value*)
	tCtr_OutlVE_RT_In.Y_min_cust			:= -1.0;	(*"customized" Y-Min at the current moment (The existing Y-Min parameter is the global minimum. To have an effect Y_min_cust needs to be > the parameter | -1.0 = function not used*)
	tCtr_OutlVE_RT_In.Y_max_cust			:=  1.0;	(*"customized" Y-Max at the current moment (The existing Y-Max parameter is the global maximum. To have an effect Y_max_cust needs to be < the parameter | 1.0 = function not used*)
	tCtr_OutlVE_RT_In.StepperMode			:= FALSE;	(* TRUE = use PWM-Mode (standard mode until 4.10) | FALSE = use continuous servo drive *)

END_PROGRAM
```

### Program Logical/Ventilation/Ctr_OutVRDP (IEC, version 4.11.0) - controller engine room differential pressure with outlet ventilation fan(s)
